FUNCTION_BLOCK "SINA_PARA_S"   // FB287, SCL
TITLE = 'one parameter exchange between SINAMICS and S7'
{ S7_Optimized_Access := 'TRUE' }
AUTHOR : DRVDPS7
FAMILY : DRIVES
NAME : SINA_PAS
VERSION : 5.0
// Copyright (C) Siemens AG 2012. All Rights Reserved. Confidential
// --------------------------------------------------------------------------- 
// SINA_PARA_S: Austausch eines beliebigen Parameter zwischen SINAMICS S120/G120 <-> S7
// -------------------------------------------------------------------------- Ersteller: J.B. Typical Team               Datum:  25.06.14        Vers.:3.0
//     Übernahme vom SINA_PARA Verion 2.9 und Abänderung zu SINA_PARA_S
//     Austausch nur noch eines Parameters
// 
// Änderung:  J.B. Typical Team                       08.07.14              3.1
//     Fehlerkorrektur und Initialisierung 
//     Änderung
// Änderung:  J.B. Typical Team                       30.07.14              4.0
//     Festlegung auf einheitlicher neuer Version 4.0
// 
// Änderung:  G.F. Typical Team                       20.05.15              4.1
//     Fehler bei der Umrechnung der Parameterwerte behoben
// 
// Änderung:  G.F. Typical Team                       15.09.15              4.2
//     Defaultwert des Parameters AxisNo von 0 auf 1 geändert
// 
// Änderung:  G.F. Typical Team                       06.10.15              4.3
//     Defaultwert des Parameters Done von 0 auf 1 geändert
// 
// Änderung:  J.B. Typical Team                       08.12.15              4.4
//     1. Wenn beim Parameter "Lesen" ein Fehler zurück gemeldet wird, 
//     soll das "Schreiben" abgebrochen werden
// 
//     2. Für den Datentyp DWORD mit/ohne Vorzeichen neuer Ablageort
//     (statt REAL nun DINT)
// 
//     3. Neue Ausgangsvariable Ready = Lesen/Schreiben der Parameter
//     abgeschlossen
// 
//     4. Austauch der Parameter kann jetzt abgebrochen werden
// 
//     5. Warnung durch Initialisierung elimininiert
// 
//     6. Eingang Laddr in hardwareId umbenannt
// 
// Änderung:  G.F. Typical Team                       24.11.16              4.5
//     - Fehlerausgabe bei unbekannten Datentyp (ErrorId := 5)
//     - Datentyp 10 (OctetString) wird unterstützt
//     - Datentyp 13 (TimeDifference) wird unterstützt
//     - Fehler bei Auftrag abbrechen behoben
// 
// Änderung:  G.F. Typical Team                       11.01.17              5.0
//     - Festlegung auf einheitlicher neuer Version 5.0 
// 
// Bibliothek V7
// Funktion: Austausch eines beliebigen Parameter zwischen SINAMICS S120/G120 <-> S7
// ********************************************************************************************************************************************************
// ************************************************************************FB283***************************************************************************
// ********************************************************************************************************************************************************
   VAR_INPUT
      Start : Bool := 0;   // Start command for read or write parameter / 0-->1 Start des gewählten azyklischen Auftrags
      ReadWrite : Bool := 0;   // Type of job 0 = read parameter, 1 = write parameter / 0 = Lesen; 1 = Schreiben
      Parameter : Int := 1;   // Number of parameter (number 1..65535) / Parameternummer
      Index : Int := 0;   // Subindex (number 0..65535) / Subindex (Number 1..65535)
      ValueWrite1 : Real := 0.0;   // Value of the write parameter (byte, word, float) / Schreibwert vom Typ REAL
      ValueWrite2 : DInt := 0;   // Value of the write parameter (dint) / Schreibwert vom Typ DINT32
      AxisNo : Byte := 16#01;   // Object ID of drive / Antriebsnummer
      hardwareId : HW_IO := 0;   // Configured diagnosis address of the module (DEC) for WRREC and RDREC Output variables / Hardware Identifer des Modul Acces Points / Istwertslots des zyklsichen Telegramms
   END_VAR
   VAR_OUTPUT
      Ready : Bool := 0;   // Read or write parameter order ready / Bereitschaftsrückmeldung für den Betrieb mit LAcycCom Bausteinen
      Busy : Bool := 0;   // Mode of operation is explained
      Done : Bool := 1;   // Mode of operation without mistake finishes
      ValueRead1 : Real := 0.0;   // Value of the read parameter (byte, word, float) / Gelesener Wert im Format REAL
      ValueRead2 : DInt := 0;   // Value of the read parameter (dint) / Gelesener Wert im Format DINT32
      Format : Byte := 16#00;   // Format of the value (Format 0x40..0x44) / Rückmeldung des Formats des gelesenen Parameters
      ErrorNo : Word := 16#0000;   // Error number (see table below) / Fehlernummer nach Profidrive Profil
      Error : Bool := 0;   // Error or faults are active / 1 = Anzeige eines aufgetretenen Fehlers
      ErrorId : DWord := 0;   // Mode of operation disturbance
      DiagId : Word := 16#0000;   // Extended communication error Static variables / Rückmeldeausgang der Systemfunktionen im Fehlerfall
   END_VAR
   VAR
      sbWrError : Bool := 0;   // Error when writing with SFB WRREC
      sbWrDone : Bool := 0;   // Data record written with SFB WRREC
      sbRdError : Bool := 0;   // Error when reading with SFB RDREC
      sbWrBusy : Bool := 0;   // Write Task busy SFB 53 WRREC sind beschäftigt
      sbRdBusy : Bool := 0;   // Read Task busy SFB 52 RDREC sind beschäftigt
      sbWrStart : Bool := 0;   // Start write job
      sbRdStart : Bool := 0;   // Start read job
      sbWrStart1 : Bool := 0;   // Start write job (first part of write commando)
      sbRdStart1 : Bool := 0;   // Start read job (first part of read commando)
      sbWrStart2 : Bool := 0;   // Start write job (second part of write commando)
      sbRdStart2 : Bool := 0;   // Start read job (second part of read commando)
      sbStart : Bool := 0;   // Positive edge of Start commando
      sbReady : Bool := 0;   // Positive edge of Ready
      sbRead : Bool := 0;   // Commando "Read"
      sbWrite : Bool := 0;   // Commando "Write"
      sbParaNo : Bool := 0;   // The count of parameter are Okay
      sbBusy : Bool := 0;   // Mode of operation is explained
      sbError : Bool := 0;   // Error or faults are active
      sbDone : Bool := 0;   // Job finished
      syFormat : Byte := 16#00;   // Format of the value (Format 0x40..0x44)
      syAxisNo : Byte := 0;   // Antriebsobjekt ID
      siReqRef : Int := 0;   // Reference number of request
      siErrorId : Int := 0;   // Function block fault Id
      siErrorCount : Int := 0;   // temporary error counter of retry job
      siMaxErrCount : Int := 12500;   // max. temporary error counter
      swParaError : Word := WORD#16#0000;   // Error of parameter
      sxReqParaMulti : Struct   // Telegramm for request/change parameter value, multi-parameter
         sxHeader : Struct   // Request header
            syReqRef : Byte := 16#00;   // Request reference (Request ID, mirrored in response)
            syReqId : Byte := 16#01;   // Request ID 0x1=Read
            syAxisNo : Byte := 16#00;   // Axis (0x0=Axis A | 0x1=Axis B)
            syParaNo : Byte := 16#00;   // No. of parameters (DEC: for single parameters=1)
         END_STRUCT;
         sxParaAdress : Struct   // Parameter address
            syAttr : Byte := 16#10;   // Attribute of parameters (0x10=Value, 0x30=Text)
            syElemNo : Byte := 16#01;   // No. of elements (DEC: for single elements=1)
            siParaNo : Int := 0;   // Number of parameter (Number 1..65535)
            siIndex : Int := 0;   // Subindex (Number 1..65535)
         END_STRUCT;
      END_STRUCT;
      sxChaParaMulti : Struct   // Telegramm for change parameter value, multi-parameter
         sxHeader : Struct   // Request header
            syReqRef : Byte := 16#00;   // Request reference (Request ID, mirrored in response)
            syReqId : Byte := 16#02;   // Request ID 0x2=Write
            syAxisNo : Byte := 16#00;   // Axis (0x0=Axis A | 0x1=Axis B)
            syParaNo : Byte := 16#00;   // No. of parameters (DEC: for single parameters=1)
         END_STRUCT;
         sxData : Array[1..12] of Byte;   // Parameter address (Attribute/Value (BYTE), Number of Elements (BYTE), Parameter number (2 BYTES), Subindex (2 BYTES),Parameter value (Format/Error (BYTE), Number of Values/Value of Error (BYTE), Value (BYTE or WORD or DWORD)
      END_STRUCT;
      sxRespParaMulti : Struct   // Telegramm for response parameter value, multi-parameter
         sxHeader : Struct   // Request header
            syReqRef : Byte := 16#00;   // Request reference (Request ID, mirrored in response)
            syReqId : Byte := 16#00;   // Request ID (0x1=Read | 0x2=Write)
            syAxisNo : Byte := 16#00;   // Axis (0x0=Axis A | 0x1=Axis B)
            syParaNo : Byte := 16#00;   // No. of parameters (DEC: for single parameters=1)
         END_STRUCT;
         sxData : Array[1..6] of Byte;   // Parameter value (Format/Error (BYTE), Number of Values/Value of Error (BYTE), Value (BYTE or WORD or DWORD)
      END_STRUCT;
      RDREC_1 : RDREC;
      WRREC_1 : WRREC;
      siLenHeader : Int := 4;   // Length of telegram of header
      siLenParaMulti : Int := 6;   // Length of telegram of data for request and response
      siLenChaPara : Int := 12;   // Length of telegram of data for change parameter Temporary variables
   END_VAR
   VAR_TEMP
      piCount : Int;   // Freely available counter variable
      piPointer : Int;   // Freely available pointer array variable
      piLenTele : Int;   // Length of telegram of buffer
      piRetSFC : Int;   // Status for fault analysis
      pwWordHigh : Word;   // Help variable of word
      pwWordLow : Word;   // Help variable of word
      pwWord1 : Word;   // Help variable of word
      pwWord2 : Word;   // Help variable of word
      pdDWordHigh : DWord;   // Help variable of dword
      pdDWordLow : DWord;   // Help variable of dword
      pdStatus : DWord;   // Status[1] = Error => Status[2] Error Decode + Status[3] Error Code
      pbValidSFB : Bool;   // Status SFB
      piLenSFB : UInt;   // Status length for SFB call
      pwErrorNo : Word;   // Error number
   END_VAR
BEGIN

   //=============================================================================
   //SIEMENS AG
   //(c)Copyright 2017 All Rights Reserved
   //-----------------------------------------------------------------------------
   // Library: DriveLib
   // Tested with: S7-1516-3 PN/DP V1.8
   // Engineering: TIA Portal V14
   // Restrictions: -
   // Requirements: S7-1200 / S7-1500
   // Functionality: read and write one parameter from/to a Sinamics
   //
   //=============================================================================

   // Auftrag "Parameter lesen" bzw. Auftrag "Parameter schreiben" wird nicht mehr ausgeführt
   IF NOT #sbBusy THEN
     #sbParaNo := TRUE;
     #syAxisNo := #AxisNo;
   END_IF;

   // Starten 
   IF #Start AND NOT #sbStart AND NOT #sbBusy THEN

     #sbReady := False;
     #sbError := False;
     #sbBusy := False;

     // Auftrag "Parameter lesen" erkennen
     IF NOT #ReadWrite THEN
       #sbRead := True;
       #sbWrStart := True;
       #sbRdStart := False;

       #sbWrite := False;
       #sbWrStart1 := False;
       #sbRdStart1 := False;
       #sbWrStart2 := False;
       #sbRdStart2 := False;

       // Referenzauftragsnummer erzeugen
       #siReqRef := #siReqRef + 1;

       // bei Überschreitung wieder zurücksetzen und von vorne (Wertebereich von 0-255)
       IF #siReqRef > 255 THEN
         #siReqRef := 0;
       END_IF;

       // Auftrag "Parameter schreiben" erkennen
     ELSE
       #sbWrite := True;
       #sbWrStart1 := True;
       #sbRdStart1 := False;
       #sbWrStart2 := False;
       #sbRdStart2 := False;

       #sbRead := False;
       #sbWrStart := False;
       #sbRdStart := False;

       // Referenzauftragsnummer erzeugen
       #siReqRef := #siReqRef + 1;

       // bei Überschreitung wieder zurücksetzen und von vorne (Wertebereich von 0-255)
       IF #siReqRef > 255 THEN
         #siReqRef := 0;
       END_IF;
     END_IF;

     // Fehler 4 und 5 wieder zurücknehmen
     IF (#siErrorId = 4) OR (#siErrorId = 5) THEN
       #sbError := False;
       #siErrorId := 0;
     END_IF;
   END_IF;

   // "Start commando" Flanke merken
   #sbStart := #Start;

   // Abbrechen
   IF NOT #Start THEN

     #siErrorCount := 0;
     // Schreib - oder Lesevorgang abbrechen
     #sbRead := False;
     #sbWrStart := False;
     #sbRdStart := False;

     #sbWrite := False;
     #sbWrStart1 := False;
     #sbRdStart1 := False;
     #sbWrStart2 := False;
     #sbRdStart2 := False;

     // Auftag ist noch beschäftigt => Fehler ausgeben
     IF #sbBusy THEN
       #sbError := True;
       #siErrorId := 4;
       #sbBusy := False;
     END_IF;
   END_IF;


   // Auftrag "Parameter lesen" wurde ausgelöst
   IF #sbParaNo AND #sbRead AND NOT #sbWrite THEN

     // Auftrag "Parameter lesen" vorbereiten und abschicken
     IF #sbWrStart THEN

       // Ablöschen des Sendepuffers
       // Parameternummer des Parameters 
       #sxReqParaMulti.sxParaAdress.siParaNo := 0;

       // Subindex des Parameters
       #sxReqParaMulti.sxParaAdress.siIndex := 0;

       // Auftrags-HEADER erstellen
       // Auftragsreferenz
       #sxReqParaMulti.sxHeader.syReqRef := INT_TO_BYTE(#siReqRef);

       // Auftragskennung 0x01=Request Parameters
       #sxReqParaMulti.sxHeader.syReqId := B#16#01;

       // Achse
       #sxReqParaMulti.sxHeader.syAxisNo := #syAxisNo;

       // Anzahl Parameter        
       #sxReqParaMulti.sxHeader.syParaNo := B#16#01;

       // Auftrags-PARAMETERADRESSE erstellen
       // Parameternummer des Parameters                                
       #sxReqParaMulti.sxParaAdress.siParaNo := #Parameter;

       // Subindex des Parameters
       #sxReqParaMulti.sxParaAdress.siIndex := #Index;

       // SCHREIBEN AZYKLISCH
       #piLenTele := #siLenHeader + #siLenParaMulti;
       #WRREC_1(REQ := True,                                // Startimpuls
                ID := #hardwareId,                         // Diagnoseadresse
                INDEX := 47,                                  // Rahmentyp
                LEN := INT_TO_UINT(#piLenTele),             // maximale Länge
                DONE => #sbWrDone,                           // Schreibauftrag beendet
                BUSY => #sbWrBusy,                           // Slave beschäftigt
                ERROR => #sbWrError,                          // Fehler beim Schreiben
                STATUS => #pdStatus,                           // Status[1] = Error => Status[2] Error Decode + Status[3] Error Code
                RECORD := #sxReqParaMulti);                    // Zeiger auf zu schreibenen Datensatzes

       // Ausgänge setzen
       #sbBusy := #sbWrBusy;
       #sbDone := #sbWrDone;

       // Fehler auswerten
       IF #sbWrError THEN

         // Fehlerstatus aus dem Doppelwort filtern und weitergeben                
         #pwWord1 := DWORD_TO_WORD(SHR(IN := (#pdStatus AND DW#16#FFFF00), N := 8));

         // Fehlerstatus setzen
         #siErrorId := 3;
         #DiagId := #pwWord1;

         //Temporärer Fehler: #pdStatus = 80A7, 80B5, 80C0, 80C1, 80C2, 80C3 oder 80C4 zulassen und nocheinmal versuchen
         IF NOT (#pwWord1 = DW#16#80A7) AND NOT (#pwWord1 = DW#16#80B5) AND NOT (#pwWord1 = DW#16#80C0) AND
           NOT (#pwWord1 = DW#16#80C1) AND NOT (#pwWord1 = DW#16#80C2) AND NOT (#pwWord1 = DW#16#80C3) AND
           NOT (#pwWord1 = DW#16#80C4) THEN

           // Wiederholungsauftrag wieder zurücknehmen 
           #sbWrStart := False;
           #sbRdStart := False;
           #sbRead := False;

           // Fehler ausgeben 
           #sbError := #sbWrError;

         ELSE
           // Fehlerwiederholauftrag ??                   
           IF #siErrorCount = #siMaxErrCount THEN

             // Wiederholungsauftrag wieder zurücknehmen
             #sbWrStart := False;
             #sbRdStart := False;
             #sbRead := False;

             //Fehlerzähler zurücksetzen
             #siErrorCount := 0;


             // Fehler ausgeben 
             #sbError := #sbWrError;

             // nix tun bis Zähler überläuft
           ELSE
             #siErrorCount := #siErrorCount + 1;
           END_IF;
         END_IF;

         // kein Fehler beim SCHEIBEN AZYKLISCH und Auftrag fertig 
       ELSIF NOT #sbWrBusy AND #sbWrDone THEN

         // Fehlerkennung zurücknehmen
         IF #siErrorId = 3 THEN
           #siErrorId := 0;
           #sbError := False;
         END_IF;

         #DiagId := W#16#00;

         // Schreibauftrag fertig melden und Leseantrag anstossen
         #sbWrStart := False;
         #sbRdStart := True;
       END_IF;
     END_IF; // Auftrag "Parameter lesen" vorbereiten und abschicken

     // vom Auftrag "Parameter lesen" die Antwort abwarten und dann auswerten
     IF #sbRdStart THEN

       // Ablöschen des Empfangspuffers
       #sxRespParaMulti.sxHeader.syReqRef := B#16#00;
       #sxRespParaMulti.sxHeader.syReqId := B#16#00;
       #sxRespParaMulti.sxHeader.syAxisNo := B#16#00;
       #sxRespParaMulti.sxHeader.syParaNo := B#16#00;

       FOR #piCount := 1 TO #siLenParaMulti DO
         #sxRespParaMulti.sxData[#piCount] := B#16#00;
       END_FOR;

       // LESEN AZYKLISCH
       #piLenTele := #siLenHeader + #siLenParaMulti;
       #RDREC_1(REQ := True,                                // Startimpuls
                ID := #hardwareId,                         // Diagnoseadresse        
                INDEX := 47,                                  // Rahmentyp           
                MLEN := INT_TO_UINT(#piLenTele),             // maximale Länge
                VALID => #pbValidSFB,                         // neuer Datensatz empfangen und gültig   
                BUSY => #sbRdBusy,                           // Slave beschäftigt
                ERROR => #sbRdError,                          // Fehler beim Schreiben
                STATUS => #pdStatus,                           // Status[1] = Error => Status[2] Error Decode + Status[3] Error Code 
                LEN => #piLenSFB,                           // Länge des gelesenen Datensatzes
                RECORD := #sxRespParaMulti);                   // Zeiger auf gelesenen Datensatz

       // Ausgänge setzen
       #sbBusy := #sbRdBusy;
       #sbDone := #pbValidSFB;

       // Fehler auswerten
       IF #sbRdError THEN
         // Fehlerstatus aus dem Doppelwort filtern und weitergeben                
         #pwWord1 := DWORD_TO_WORD(SHR(IN := (#pdStatus AND DW#16#FFFF00), N := 8));

         // Fehlerstatus setzen
         #siErrorId := 3;
         #DiagId := #pwWord1;

         //Temporärer Fehler: #pdStatus = 80A7, 80B5, 80C0, 80C1, 80C2, 80C3 oder 80C4 zulassen und nocheinmal versuchen
         IF NOT (#pwWord1 = DW#16#80A7) AND NOT (#pwWord1 = DW#16#80B5) AND NOT (#pwWord1 = DW#16#80C0) AND
           NOT (#pwWord1 = DW#16#80C1) AND NOT (#pwWord1 = DW#16#80C2) AND NOT (#pwWord1 = DW#16#80C3) AND
           NOT (#pwWord1 = DW#16#80C4) THEN

           // Wiederholungsauftrag wieder zurücknehmen  
           #sbWrStart := False;
           #sbRdStart := False;
           #sbRead := False;

           // Fehler ausgeben 
           #sbError := #sbRdError;

         ELSE
           // Fehlerwiederholauftrag ??                   
           IF #siErrorCount = #siMaxErrCount THEN

             // Wiederholungsauftrag wieder zurücknehmen
             #sbWrStart := False;
             #sbRdStart := False;
             #sbRead := False;

             //Fehlerzähler zurücksetzen
             #siErrorCount := 0;


             // Fehler ausgeben 
             #sbError := #sbRdError;

             // nix tun bis Zähler überläuft
           ELSE
             #siErrorCount := #siErrorCount + 1;
           END_IF;
         END_IF;

         // Fehler : die Auftragsreferenz der Antwort übertimmt nicht mit der Auftragsreferenz der Anfrage überein
       ELSIF NOT (#siReqRef = BYTE_TO_INT(#sxRespParaMulti.sxHeader.syReqRef)) AND NOT #sbRdBusy AND #pbValidSFB THEN
         #siErrorId := 1;
         #sbError := True;
         #sbDone := False;

         // Wiederholungsauftrag wieder zurücknehmen  
         #sbWrStart := False;
         #sbRdStart := False;
         #sbRead := False;

         // Fehler : falsche Auftragskennung zurück erhalten    
       ELSIF NOT (#sxRespParaMulti.sxHeader.syReqId = B#16#81 OR #sxRespParaMulti.sxHeader.syReqId = B#16#01) AND
         NOT #sbRdBusy AND #pbValidSFB THEN
         #siErrorId := 1;
         #sbError := True;
         #sbDone := False;

         // Wiederholungsauftrag wieder zurücknehmen  
         #sbWrStart := False;
         #sbRdStart := False;
         #sbRead := False;

         // Fehler : die angeforderte Anzahl Parameter entspricht nicht der übermittelten Anzahl Parameter überein
       ELSIF NOT (#sxRespParaMulti.sxHeader.syParaNo = B#16#01) AND NOT #sbRdBusy AND #pbValidSFB THEN
         #siErrorId := 1;
         #sbError := True;
         #sbDone := False;

         // Wiederholungsauftrag wieder zurücknehmen  
         #sbWrStart := False;
         #sbRdStart := False;
         #sbRead := False;

         // Fehler : die Achse entspricht nicht der übergebenen Achse
       ELSIF NOT (#syAxisNo = #sxRespParaMulti.sxHeader.syAxisNo) AND NOT #sbRdBusy AND #pbValidSFB THEN
         #siErrorId := 1;
         #sbError := True;
         #sbDone := False;

         // Wiederholungsauftrag wieder zurücknehmen  
         #sbWrStart := False;
         #sbRdStart := False;
         #sbRead := False;

         // kein Fehler beim LESEN AZYKLISCH und Auftrag fertig 
       ELSIF NOT #sbRdBusy AND #pbValidSFB THEN

         // die angefragten Parameter auswerten und im Puffer abspeichern

         // ermitteltes Format des Parameters abspeichern
         #syFormat := #sxRespParaMulti.sxData[1];

         // Format = Error ? = > gesendeter Parameter fehlerhaft
         IF (BYTE_TO_INT(#sxRespParaMulti.sxData[1]) = 68) THEN

           // Format = Error, zwei Bytes zu übermittelten Fehlernummer zusammenfassen
           #pwWordHigh := SHL(IN := BYTE_TO_WORD(#sxRespParaMulti.sxData[3]), N := 8);
           #pwWordLow := BYTE_TO_WORD(#sxRespParaMulti.sxData[4]);

           #sbError := True;

           // ermittelte Fehlernummer im Puffer abspeichern
           #ErrorNo := #pwWordHigh XOR #pwWordLow;

           // Die Fehlerhaftigkeit des erkannten Parameter in der Fehlernummer eintragen   
           #swParaError := #swParaError OR W#16#01;

           // Format = Byte ? = > gesendeter Parameter ein Byte lang ohne Vorzeichen
         ELSIF (#sxRespParaMulti.sxData[1] = B#16#41) OR (#sxRespParaMulti.sxData[1] = B#16#05) THEN

           // ermittelter Parameterwert eintragen (Byte) 
           #ValueRead1 := USINT_TO_REAL(BYTE_TO_USINT(#sxRespParaMulti.sxData[3]));
           #ValueRead2 := 0;

           // ermittelte Fehlernummer im Puffer zurücksetzen
           #ErrorNo := W#16#00;

           // Die Fehlerhaftigkeit des erkannten Parameter in der Fehlernummer löschen   
           #swParaError := #swParaError AND W#16#FFFE;

           // Format = Byte ? = > gesendeter Parameter ein Byte lang mit Vorzeichen
         ELSIF (#sxRespParaMulti.sxData[1] = B#16#02) THEN

           // ermittelter Parameterwert eintragen (Byte) 
           #ValueRead1 := SINT_TO_REAL(BYTE_TO_SINT(#sxRespParaMulti.sxData[3]));
           #ValueRead2 := 0;

           // ermittelte Fehlernummer im Puffer zurücksetzen
           #ErrorNo := W#16#00;

           // Die Fehlerhaftigkeit des erkannten Parameter in der Fehlernummer löschen   
           #swParaError := #swParaError AND W#16#FFFE;

           // Format = Word ? = > gesendeter Parameter zwei Bytes lang ohne Vorzeichen
         ELSIF (#sxRespParaMulti.sxData[1] = B#16#42) OR (#sxRespParaMulti.sxData[1] = B#16#06)
           OR (#sxRespParaMulti.sxData[1] = B#16#0A) THEN

           // Format = Word, zwei Bytes zu übermitteltem Parameterwert zusammenfassen
           #pwWordHigh := SHL(IN := BYTE_TO_WORD(#sxRespParaMulti.sxData[3]), N := 8);
           #pwWordLow := BYTE_TO_WORD(#sxRespParaMulti.sxData[4]);
           #pwWord1 := #pwWordHigh XOR #pwWordLow;

           // ermittelter Parameterwert eintragen (Word)
           #ValueRead1 := UINT_TO_REAL(WORD_TO_UINT(#pwWord1));
           #ValueRead2 := 0;

           // ermittelte Fehlernummer im Puffer zurücksetzen
           #ErrorNo := W#16#00;

           // Die Fehlerhaftigkeit des erkannten Parameter in der Fehlernummer löschen   
           #swParaError := #swParaError AND W#16#FFFE;

           // Format = Word ? = > gesendeter Parameter zwei Bytes lang mit Vorzeichen
         ELSIF (#sxRespParaMulti.sxData[1] = B#16#03) THEN

           // Format = Word, zwei Bytes zu übermitteltem Parameterwert zusammenfassen
           #pwWordHigh := SHL(IN := BYTE_TO_WORD(#sxRespParaMulti.sxData[3]), N := 8);
           #pwWordLow := BYTE_TO_WORD(#sxRespParaMulti.sxData[4]);
           #pwWord1 := #pwWordHigh XOR #pwWordLow;

           // ermittelter Parameterwert eintragen (Word)
           #ValueRead1 := INT_TO_REAL(WORD_TO_INT(#pwWord1));
           #ValueRead2 := 0;

           // ermittelte Fehlernummer im Puffer zurücksetzen
           #ErrorNo := W#16#00;

           // Die Fehlerhaftigkeit des erkannten Parameter in der Fehlernummer löschen   
           #swParaError := #swParaError AND W#16#FFFE;

           // Format = Double Word ? = > gesendeter Parameter vier Bytes lang ohne Vorzeichen
         ELSIF (#sxRespParaMulti.sxData[1] = B#16#43) OR (#sxRespParaMulti.sxData[1] = B#16#07) OR
           (#sxRespParaMulti.sxData[1] = B#16#0D) THEN

           // Format = Double Word, vier Bytes zu übermitteltem Parameterwert zusammenfassen
           #pwWordHigh := SHL(IN := BYTE_TO_WORD(#sxRespParaMulti.sxData[3]), N := 8);
           #pwWordLow := BYTE_TO_WORD(#sxRespParaMulti.sxData[4]);
           #pwWord1 := #pwWordHigh XOR #pwWordLow;

           #pwWordHigh := SHL(IN := BYTE_TO_WORD(#sxRespParaMulti.sxData[5]), N := 8);
           #pwWordLow := BYTE_TO_WORD(#sxRespParaMulti.sxData[6]);
           #pwWord2 := #pwWordHigh XOR #pwWordLow;

           #pdDWordHigh := SHL(IN := WORD_TO_DWORD(#pwWord1), N := 16);
           #pdDWordLow := WORD_TO_DWORD(#pwWord2);

           // ermittelter Parameterwert eintragen (Word)
           #ValueRead1 := 0.0;
           #ValueRead2 := DWORD_TO_DINT(#pdDWordHigh XOR #pdDWordLow);

           // ermittelte Fehlernummer im Puffer zurücksetzen
           #ErrorNo := W#16#00;

           // Die Fehlerhaftigkeit des erkannten Parameter in der Fehlernummer löschen   
           #swParaError := #swParaError AND W#16#FFFE;

           // Format = Double Word ? = > gesendeter Parameter vier Bytes lang mit Vorzeichen
         ELSIF (#sxRespParaMulti.sxData[1] = B#16#04) THEN

           // Format = Double Word, vier Bytes zu übermitteltem Parameterwert zusammenfassen
           #pwWordHigh := SHL(IN := BYTE_TO_WORD(#sxRespParaMulti.sxData[3]), N := 8);
           #pwWordLow := BYTE_TO_WORD(#sxRespParaMulti.sxData[4]);
           #pwWord1 := #pwWordHigh XOR #pwWordLow;

           #pwWordHigh := SHL(IN := BYTE_TO_WORD(#sxRespParaMulti.sxData[5]), N := 8);
           #pwWordLow := BYTE_TO_WORD(#sxRespParaMulti.sxData[6]);
           #pwWord2 := #pwWordHigh XOR #pwWordLow;

           #pdDWordHigh := SHL(IN := WORD_TO_DWORD(#pwWord1), N := 16);
           #pdDWordLow := WORD_TO_DWORD(#pwWord2);

           // ermittelter Parameterwert eintragen (Word)
           #ValueRead1 := 0.0;
           #ValueRead2 := DWORD_TO_DINT(#pdDWordHigh XOR #pdDWordLow);

           // ermittelte Fehlernummer im Puffer zurücksetzen
           #ErrorNo := W#16#00;

           // Die Fehlerhaftigkeit des erkannten Parameter in der Fehlernummer löschen   
           #swParaError := #swParaError AND W#16#FFFE;

           // Format = Double Word ? = > gesendeter Parameter vier Bytes lang (FloatingPoint)
         ELSIF (#sxRespParaMulti.sxData[1] = B#16#08) THEN

           // Format = Double Word, vier Bytes zu übermitteltem Parameterwert zusammenfassen
           #pwWordHigh := SHL(IN := BYTE_TO_WORD(#sxRespParaMulti.sxData[3]), N := 8);
           #pwWordLow := BYTE_TO_WORD(#sxRespParaMulti.sxData[4]);
           #pwWord1 := #pwWordHigh XOR #pwWordLow;

           #pwWordHigh := SHL(IN := BYTE_TO_WORD(#sxRespParaMulti.sxData[5]), N := 8);
           #pwWordLow := BYTE_TO_WORD(#sxRespParaMulti.sxData[6]);
           #pwWord2 := #pwWordHigh XOR #pwWordLow;

           #pdDWordHigh := SHL(IN := WORD_TO_DWORD(#pwWord1), N := 16);
           #pdDWordLow := WORD_TO_DWORD(#pwWord2);

           // ermittelter Parameterwert eintragen (Word)
           #ValueRead1 := DWORD_TO_REAL(#pdDWordHigh XOR #pdDWordLow);
           #ValueRead2 := 0;

           // ermittelte Fehlernummer im Puffer zurücksetzen
           #ErrorNo := W#16#00;

           // Die Fehlerhaftigkeit des erkannten Parameter in der Fehlernummer löschen   
           #swParaError := #swParaError AND W#16#FFFE;

           // Unbekanter Datentyp
         ELSE

           #siErrorId := 5;
           #sbError := True;
           #sbDone := False;
           // Die Fehlerhaftigkeit des erkannten Parameter in der Fehlernummer eintragen   
           #swParaError := #swParaError OR W#16#01;

         END_IF;

         // Fehlerkennung zurücknehmen
         IF (#siErrorId = 3) OR (#siErrorId = 1) THEN
           #siErrorId := 0;
           #sbError := False;
         END_IF;

         #DiagId := W#16#00;

         // Auftrag : Parameter lesen ist abgeschlossen
         #sbRdStart := False;
         #sbRead := False;
       END_IF; // kein Fehler beim LESEN AZYKLISCH und Auftrag fertig 
     END_IF; // vom Auftrag "Parameter lesen" die Antwort abwarten und dann auswerten 
   END_IF; // Auftrag "Parameter lesen" wurde ausgelöst

   // Auftrag "Parameter schreiben" wurde ausgelöst
   IF #sbParaNo AND NOT #sbRead AND #sbWrite THEN

     // Auftrag "Parameter schreiben" bzw. "ändern" besteht aus zwei Aufträgen
     // 1. Teilauftrag "Parameter lesen"
     // 2. Teilauftrag "Parameter schreiben bzw. ändern"

     // 1. Teilauftrag "Parameter lesen" vorbereiten und abschicken
     IF #sbWrStart1 THEN

       // Ablöschen des Sendepuffers
       // Parameternummer des Parameters 
       #sxReqParaMulti.sxParaAdress.siParaNo := 0;

       // Subindex des Parameters
       #sxReqParaMulti.sxParaAdress.siIndex := 0;

       // Auftrags-HEADER erstellen
       // Auftragsreferenz
       #sxReqParaMulti.sxHeader.syReqRef := INT_TO_BYTE(#siReqRef);

       // Auftragskennung 0x01=Request Parameters
       #sxReqParaMulti.sxHeader.syReqId := B#16#01;

       // Achse
       #sxReqParaMulti.sxHeader.syAxisNo := #syAxisNo;

       // Anzahl Parameter        
       #sxReqParaMulti.sxHeader.syParaNo := B#16#01;

       // Auftrags-PARAMETERADRESSE erstellen
       // Parameternummer des Parameters                                
       #sxReqParaMulti.sxParaAdress.siParaNo := #Parameter;

       // Subindex des Parameters
       #sxReqParaMulti.sxParaAdress.siIndex := #Index;

       // SCHREIBEN AZYKLISCH
       #piLenTele := #siLenHeader + #siLenParaMulti;
       #WRREC_1(REQ := True,                                // Startimpuls
                ID := #hardwareId,                         // Diagnoseadresse
                INDEX := 47,                                  // Rahmentyp
                LEN := INT_TO_UINT(#piLenTele),             // maximale Länge
                DONE => #sbWrDone,                           // Schreibauftrag beendet
                BUSY => #sbWrBusy,                           // Slave beschäftigt
                ERROR => #sbWrError,                          // Fehler beim Schreiben
                STATUS => #pdStatus,                           // Status[1] = Error => Status[2] Error Decode + Status[3] Error Code
                RECORD := #sxReqParaMulti);                    // Zeiger auf zu schreibenen Datensatz

       // Ausgänge setzen
       #sbBusy := #sbWrBusy;
       #sbDone := #sbWrDone;

       // Fehler auswerten
       IF #sbWrError THEN

         // Fehlerstatus aus dem Doppelwort filtern und weitergeben                
         #pwWord1 := DWORD_TO_WORD(SHR(IN := (#pdStatus AND DW#16#FFFF00), N := 8));

         // Fehlerstatus setzen
         #siErrorId := 3;
         #DiagId := #pwWord1;

         //Temporärer Fehler: #pdStatus = 80A7, 80B5, 80C0, 80C1, 80C2, 80C3 oder 80C4 zulassen und nocheinmal versuchen
         IF NOT (#pwWord1 = DW#16#80A7) AND NOT (#pwWord1 = DW#16#80B5) AND NOT (#pwWord1 = DW#16#80C0) AND
           NOT (#pwWord1 = DW#16#80C1) AND NOT (#pwWord1 = DW#16#80C2) AND NOT (#pwWord1 = DW#16#80C3) AND
           NOT (#pwWord1 = DW#16#80C4) THEN

           // Wiederholungsauftrag wieder zurücknehmen
           #sbWrStart1 := False;
           #sbRdStart1 := False;
           #sbWrite := False;

           // Fehler ausgeben 
           #sbError := #sbWrError;

         ELSE
           // Fehlerwiederholauftrag ??                   
           IF #siErrorCount = #siMaxErrCount THEN

             // Wiederholungsauftrag wieder zurücknehmen
             #sbWrStart1 := False;
             #sbRdStart1 := False;
             #sbWrite := False;

             //Fehlerzähler zurücksetzen
             #siErrorCount := 0;


             // Fehler ausgeben 
             #sbError := #sbWrError;
             // nix tun bis Zähler überläuft
           ELSE
             #siErrorCount := #siErrorCount + 1;
           END_IF;
         END_IF;

         // kein Fehler beim SCHEIBEN AZYKLISCH und Auftrag fertig 
       ELSIF NOT #sbWrBusy AND #sbWrDone THEN

         // Fehlerkennung zurücknehmen
         IF (#siErrorId = 3) THEN
           #siErrorId := 0;
           #sbError := False;
         END_IF;

         #DiagId := W#16#00;

         // Schreibauftrag fertig melden und Leseantrag anstossen
         #sbWrStart1 := False;
         #sbRdStart1 := True;
       END_IF;
     END_IF; // 1. Teilauftrag "Parameter lesen" vorbereiten und abschicken

     // vom 1. Teilauftrag "Parameter lesen" die Antwort abwarten und dann auswerten
     IF #sbRdStart1 THEN

       // Ablöschen des Empfangspuffers
       #sxRespParaMulti.sxHeader.syReqRef := B#16#00;
       #sxRespParaMulti.sxHeader.syReqId := B#16#00;
       #sxRespParaMulti.sxHeader.syAxisNo := B#16#00;
       #sxRespParaMulti.sxHeader.syParaNo := B#16#00;

       FOR #piCount := 1 TO #siLenParaMulti DO
         #sxRespParaMulti.sxData[#piCount] := B#16#00;
       END_FOR;

       // LESEN AZYKLISCH
       #piLenTele := #siLenHeader + #siLenParaMulti;
       #RDREC_1(REQ := True,                                // Startimpuls
                ID := #hardwareId,                         // Diagnoseadresse        
                INDEX := 47,                                  // Rahmentyp           
                MLEN := INT_TO_UINT(#piLenTele),             // maximale Länge
                VALID => #pbValidSFB,                         // neuer Datensatz empfangen und gültig      
                BUSY => #sbRdBusy,                           // Slave beschäftigt
                ERROR => #sbRdError,                          // Fehler beim Schreiben
                STATUS => #pdStatus,                           // Status[1] = Error => Status[2] Error Decode + Status[3] Error Code 
                LEN => #piLenSFB,                           // Länge des gelesenen Datensatzes
                RECORD := #sxRespParaMulti);                   // Zeiger auf gelesenen Datensatz

       // Ausgänge setzen
       #sbBusy := #sbRdBusy;
       #sbDone := #pbValidSFB;

       // Fehler auswerten
       IF #sbRdError THEN
         // Fehlerstatus aus dem Doppelwort filtern und weitergeben                
         #pwWord1 := DWORD_TO_WORD(SHR(IN := (#pdStatus AND DW#16#FFFF00), N := 8));

         // Fehlerstatus setzen
         #siErrorId := 3;
         #DiagId := #pwWord1;

         //Temporärer Fehler: #pdStatus = 80A7, 80B5, 80C0, 80C1, 80C2, 80C3 oder 80C4 zulassen und nocheinmal versuchen
         IF NOT (#pwWord1 = DW#16#80A7) AND NOT (#pwWord1 = DW#16#80B5) AND NOT (#pwWord1 = DW#16#80C0) AND
           NOT (#pwWord1 = DW#16#80C1) AND NOT (#pwWord1 = DW#16#80C2) AND NOT (#pwWord1 = DW#16#80C3) AND
           NOT (#pwWord1 = DW#16#80C4) THEN

           // Wiederholungsauftrag wieder zurücknehmen
           #sbWrStart1 := False;
           #sbRdStart1 := False;
           #sbWrite := False;

           // Fehler ausgeben 
           #sbError := #sbRdError;

         ELSE
           // Fehlerwiederholauftrag ??                   
           IF #siErrorCount = #siMaxErrCount THEN

             // Wiederholungsauftrag wieder zurücknehmen
             #sbWrStart1 := False;
             #sbRdStart1 := False;
             #sbWrite := False;

             //Fehlerzähler zurücksetzen
             #siErrorCount := 0;


             // Fehler ausgeben 
             #sbError := #sbRdError;

             // nix tun bis Zähler überläuft
           ELSE
             #siErrorCount := #siErrorCount + 1;
           END_IF;
         END_IF;

         // Fehler : die Auftragsreferenz der Antwort übertimmt nicht mit der Auftragsreferenz der Anfrage überein
       ELSIF NOT (#siReqRef = BYTE_TO_INT(#sxRespParaMulti.sxHeader.syReqRef)) AND NOT #sbRdBusy AND #pbValidSFB THEN
         #siErrorId := 1;
         #sbError := True;
         #sbDone := False;

         // Wiederholungsauftrag wieder zurücknehmen
         #sbWrStart1 := False;
         #sbRdStart1 := False;
         #sbWrite := False;

         // Fehler : falsche Auftragskennung zurück erhalten    
       ELSIF NOT (#sxRespParaMulti.sxHeader.syReqId = B#16#81 OR #sxRespParaMulti.sxHeader.syReqId = B#16#01) AND
         NOT #sbRdBusy AND #pbValidSFB THEN
         #siErrorId := 1;
         #sbError := True;
         #sbDone := False;

         // Wiederholungsauftrag wieder zurücknehmen
         #sbWrStart1 := False;
         #sbRdStart1 := False;
         #sbWrite := False;

         // Fehler : die angeforderte Anzahl Parameter entspricht nicht der übermittelten Anzahl Parameter überein
       ELSIF NOT (#sxRespParaMulti.sxHeader.syParaNo = B#16#01) AND NOT #sbRdBusy AND #pbValidSFB THEN
         #siErrorId := 1;
         #sbError := True;
         #sbDone := False;

         // Wiederholungsauftrag wieder zurücknehmen
         #sbWrStart1 := False;
         #sbRdStart1 := False;
         #sbWrite := False;

         // Fehler : die Achse entspricht nicht der übergebenen Achse
       ELSIF NOT (#syAxisNo = #sxRespParaMulti.sxHeader.syAxisNo) AND NOT #sbRdBusy AND #pbValidSFB THEN
         #siErrorId := 1;
         #sbError := True;
         #sbDone := False;

         // Wiederholungsauftrag wieder zurücknehmen
         #sbWrStart1 := False;
         #sbRdStart1 := False;
         #sbWrite := False;

         // kein Fehler beim LESEN AZYKLISCH und Auftrag fertig 
       ELSIF NOT #sbRdBusy AND #pbValidSFB THEN

         // die angefragten Parameter auswerten und im Puffer abspeichern
         // ermitteltes Format des Parameters abspeichern
         #syFormat := #sxRespParaMulti.sxData[1];

         // Format = Error ? = > gesendeter Parameter fehlerhaft
         IF (BYTE_TO_INT(#sxRespParaMulti.sxData[1]) = 68) THEN

           // Format = Error, zwei Bytes zu übermittelten Fehlernummer zusammenfassen
           #pwWordHigh := SHL(IN := BYTE_TO_WORD(#sxRespParaMulti.sxData[3]), N := 8);
           #pwWordLow := BYTE_TO_WORD(#sxRespParaMulti.sxData[4]);

           #sbError := True;

           // ermittelte Fehlernummer im Puffer abspeichern
           #ErrorNo := #pwWordHigh XOR #pwWordLow;

           // Die Fehlerhaftigkeit des erkannten Parameter in der Fehlernummer eintragen   
           #swParaError := #swParaError OR W#16#01;

           // Format = Byte ? = > gesendeter Parameter ein Byte lang
         ELSIF (#sxRespParaMulti.sxData[1] = B#16#41) OR
           (#sxRespParaMulti.sxData[1] = B#16#02) OR (#sxRespParaMulti.sxData[1] = B#16#05) THEN

           // ermittelte Fehlernummer im Puffer zurücksetzen
           #ErrorNo := W#16#00;

           // Die Fehlerhaftigkeit des erkannten Parameter in der Fehlernummer löschen   
           #swParaError := #swParaError AND W#16#FFFE;

           // Format = Word ? = > gesendeter Parameter zwei Bytes lang
         ELSIF (#sxRespParaMulti.sxData[1] = B#16#42) OR (#sxRespParaMulti.sxData[1] = B#16#03)
           OR (#sxRespParaMulti.sxData[1] = B#16#06) OR (#sxRespParaMulti.sxData[1] = B#16#0A) THEN

           // ermittelte Fehlernummer im Puffer zurücksetzen
           #ErrorNo := W#16#00;

           // Die Fehlerhaftigkeit des erkannten Parameter in der Fehlernummer löschen   
           #swParaError := #swParaError AND W#16#FFFE;


           // Format = Double Word ? = > gesendeter Parameter vier Bytes lang
         ELSIF (#sxRespParaMulti.sxData[1] = B#16#43) OR (#sxRespParaMulti.sxData[1] = B#16#04) OR
           (#sxRespParaMulti.sxData[1] = B#16#07) OR (#sxRespParaMulti.sxData[1] = B#16#08) OR
           (#sxRespParaMulti.sxData[1] = B#16#0D) THEN

           // ermittelte Fehlernummer im Puffer zurücksetzen
           #ErrorNo := W#16#00;

           // Die Fehlerhaftigkeit des erkannten Parameter in der Fehlernummer löschen   
           #swParaError := #swParaError AND W#16#FFFE;

           // Unbekanter Datentyp
         ELSE

           #siErrorId := 5;
           #sbError := True;
           #sbDone := False;
           // Die Fehlerhaftigkeit des erkannten Parameter in der Fehlernummer eintragen   
           #swParaError := #swParaError OR W#16#01;

         END_IF;

         // Fehlerkennung zurücknehmen
         IF (#siErrorId = 3) OR (#siErrorId = 1) THEN
           #siErrorId := 0;
           #sbError := False;
         END_IF;

         #DiagId := W#16#00;

         // 1. Teilauftrag "Parameter lesen" ist abgeschlossen
         #sbRdStart1 := False;

         // einer der gesendeten Parameter ist fehlerhaft => Abbruch, kein "Parameter schreiben" erforderlich
         IF (#swParaError = W#16#00) THEN
           #sbWrStart2 := True;
         ELSE
           #sbWrStart2 := False;
         END_IF;
       END_IF; // kein Fehler beim LESEN AZYKLISCH und Auftrag fertig 
     END_IF; // vom 1. Teilauftrag "Parameter lesen" die Antwort abwarten und dann auswerten 

     // 2. Teilauftrag "Parameter schreiben bzw. ändern" vorbereiten und abschicken
     IF #sbWrStart2 THEN

       // Ablöschen des Sendepuffers            
       FOR #piCount := 1 TO #siLenChaPara DO
         // Parameteradresse und Parameterwert des Parameters 
         #sxChaParaMulti.sxData[#piCount] := B#16#00;
       END_FOR;

       // Auftrags-HEADER erstellen
       // Auftragsreferenz
       #sxChaParaMulti.sxHeader.syReqRef := INT_TO_BYTE(#siReqRef);

       // Auftragskennung 0x01=Request Parameters | 0x02=Change Parameters
       #sxChaParaMulti.sxHeader.syReqId := B#16#02;

       // Achse
       #sxChaParaMulti.sxHeader.syAxisNo := #syAxisNo;

       // Anzahl Parameter        
       #sxChaParaMulti.sxHeader.syParaNo := B#16#01;

       // Auftrags-PARAMETERADRESSE erstellen                
       // Attribute of parameters (0x10=Value, 0x30=Text)
       #sxChaParaMulti.sxData[1] := B#16#10;

       // No. of elements (DEC: for single elements=1) 
       #sxChaParaMulti.sxData[2] := B#16#01;

       // Parameternummer des Parameters                                
       #sxChaParaMulti.sxData[4] := INT_TO_BYTE(#Parameter);
       #sxChaParaMulti.sxData[3] := WORD_TO_BYTE(SHR(IN := INT_TO_WORD(#Parameter), N := 8));

       // Subindex des Parameters
       #sxChaParaMulti.sxData[6] := INT_TO_BYTE(#Index);
       #sxChaParaMulti.sxData[5] := WORD_TO_BYTE(SHR(IN := INT_TO_WORD(#Index), N := 8));

       // Auftrags-PARAMETERVALUE erstellen    
       // Format (BYTE, WORD, DWORD des Parameterwert übergeben
       #sxChaParaMulti.sxData[7] := #syFormat;

       // Number of value
       #sxChaParaMulti.sxData[8] := B#16#01;

       // Value of parameter in Bytes
       IF (#syFormat = B#16#41) OR
         (#syFormat = B#16#02) OR (#syFormat = B#16#05) THEN

         #sxChaParaMulti.sxData[9] := WORD_TO_BYTE(DWORD_TO_WORD(DINT_TO_DWORD(REAL_TO_DINT(#ValueWrite1))));
         #sxChaParaMulti.sxData[10] := 16#00;  //WORD_TO_BYTE(DWORD_TO_WORD(SHR(IN := DINT_TO_DWORD(REAL_TO_DINT(#ValueWrite1)), N := 8)));

         // Value of parameter in Word
       ELSIF (#syFormat = B#16#42) OR (#syFormat = B#16#03) OR
         (#syFormat = B#16#06) OR (#syFormat = B#16#0A) THEN

         #sxChaParaMulti.sxData[10] := WORD_TO_BYTE(DWORD_TO_WORD(DINT_TO_DWORD(REAL_TO_DINT(#ValueWrite1))));
         #sxChaParaMulti.sxData[9] := WORD_TO_BYTE(DWORD_TO_WORD(SHR(IN := DINT_TO_DWORD(REAL_TO_DINT(#ValueWrite1)), N := 8)));

         // Value of parameter in DWord    
       ELSIF (#syFormat = B#16#43) OR (#syFormat = B#16#04) OR
         (#syFormat = B#16#07) OR (#syFormat = B#16#0D) THEN

         #sxChaParaMulti.sxData[12] := WORD_TO_BYTE(DWORD_TO_WORD(DINT_TO_DWORD(#ValueWrite2)));
         #sxChaParaMulti.sxData[11] := WORD_TO_BYTE(DWORD_TO_WORD(SHR(IN := DINT_TO_DWORD(#ValueWrite2), N := 8)));
         #sxChaParaMulti.sxData[10] := WORD_TO_BYTE(DWORD_TO_WORD(SHR(IN := DINT_TO_DWORD(#ValueWrite2), N := 16)));
         #sxChaParaMulti.sxData[9] := WORD_TO_BYTE(DWORD_TO_WORD(SHR(IN := DINT_TO_DWORD(#ValueWrite2), N := 24)));


         // Value of parameter in DWord (FloatingPoint)   
       ELSIF (#syFormat = B#16#08) THEN

         #sxChaParaMulti.sxData[12] := WORD_TO_BYTE(DWORD_TO_WORD(REAL_TO_DWORD(#ValueWrite1)));
         #sxChaParaMulti.sxData[11] := WORD_TO_BYTE(DWORD_TO_WORD(SHR(IN := REAL_TO_DWORD(#ValueWrite1), N := 8)));
         #sxChaParaMulti.sxData[10] := WORD_TO_BYTE(DWORD_TO_WORD(SHR(IN := REAL_TO_DWORD(#ValueWrite1), N := 16)));
         #sxChaParaMulti.sxData[9] := WORD_TO_BYTE(DWORD_TO_WORD(SHR(IN := REAL_TO_DWORD(#ValueWrite1), N := 24)));

       END_IF;

       // SCHREIBEN AZYKLISCH
       #piLenTele := #siLenHeader + #siLenChaPara;
       #WRREC_1(REQ := True,                                // Startimpuls
                ID := #hardwareId,                         // Diagnoseadresse
                INDEX := 47,                                  // Rahmentyp
                LEN := INT_TO_UINT(#piLenTele),             // maximale Länge
                DONE => #sbWrDone,                           // Schreibauftrag beendet
                BUSY => #sbWrBusy,                           // Slave beschäftigt
                ERROR => #sbWrError,                          // Fehler beim Schreiben
                STATUS => #pdStatus,                           // Status[1] = Error => Status[2] Error Decode + Status[3] Error Code
                RECORD := #sxChaParaMulti);                    // Zeiger auf zu schreibenen Datensatzes

       // Ausgänge setzen
       #sbBusy := #sbWrBusy;
       #sbDone := #sbWrDone;

       // Fehler auswerten
       IF #sbWrError THEN
         // Fehlerstatus aus dem Doppelwort filtern und weitergeben                
         #pwWord1 := DWORD_TO_WORD(SHR(IN := (#pdStatus AND DW#16#FFFF00), N := 8));

         // Fehlerstatus setzen
         #siErrorId := 3;
         #sbError := False;
         #DiagId := #pwWord1;

         //Temporärer Fehler: #pdStatus = 80A7, 80B5, 80C0, 80C1, 80C2, 80C3 oder 80C4 zulassen und nocheinmal versuchen
         IF NOT (#pwWord1 = DW#16#80A7) AND NOT (#pwWord1 = DW#16#80B5) AND NOT (#pwWord1 = DW#16#80C0) AND
           NOT (#pwWord1 = DW#16#80C1) AND NOT (#pwWord1 = DW#16#80C2) AND NOT (#pwWord1 = DW#16#80C3) AND
           NOT (#pwWord1 = DW#16#80C4) THEN

           // Wiederholungsauftrag wieder zurücknehmen
           #sbWrStart2 := False;
           #sbRdStart2 := False;
           #sbWrite := False;

           // Fehler ausgeben 
           #sbError := #sbWrError;

         ELSE
           // Fehlerwiederholauftrag ??                   
           IF #siErrorCount = #siMaxErrCount THEN

             // Wiederholungsauftrag wieder zurücknehmen
             #sbWrStart2 := False;
             #sbRdStart2 := False;
             #sbWrite := False;

             //Fehlerzähler zurücksetzen
             #siErrorCount := 0;


             // Fehler ausgeben 
             #sbError := #sbWrError;

             // nix tun bis Zähler überläuft
           ELSE
             #siErrorCount := #siErrorCount + 1;
           END_IF;
         END_IF;

         // kein Fehler beim SCHEIBEN AZYKLISCH und Auftrag fertig 
       ELSIF NOT #sbWrBusy AND #sbWrDone THEN
         // Fehlerkennung zurücknehmen
         #DiagId := W#16#00;

         // Schreibauftrag fertig melden und Leseantrag anstossen
         #sbWrStart2 := False;
         #sbRdStart2 := True;
       END_IF;
     END_IF; // 2. Teilauftrag "Parameter schreiben bzw. ändern" vorbereiten und abschicken

     // vom 2. Teilauftrag "Parameter schreiben bzw. ändern" die Antwort abwarten und dann auswerten
     IF #sbRdStart2 THEN

       // Ablöschen des Empfangspuffers
       #sxRespParaMulti.sxHeader.syReqRef := B#16#00;
       #sxRespParaMulti.sxHeader.syReqId := B#16#00;
       #sxRespParaMulti.sxHeader.syAxisNo := B#16#00;
       #sxRespParaMulti.sxHeader.syParaNo := B#16#00;

       FOR #piCount := 1 TO #siLenParaMulti DO
         #sxRespParaMulti.sxData[#piCount] := B#16#00;
       END_FOR;

       // LESEN AZYKLISCH
       #piLenTele := #siLenHeader + #siLenParaMulti;
       #RDREC_1(REQ := True,                                // Startimpuls
                ID := #hardwareId,                         // Diagnoseadresse        
                INDEX := 47,                                  // Rahmentyp           
                MLEN := INT_TO_UINT(#piLenTele),             // maximale Länge
                VALID => #pbValidSFB,                         // neuer Datensatz empfangen und gültig   
                BUSY => #sbRdBusy,                           // Slave beschäftigt
                ERROR => #sbRdError,                          // Fehler beim Schreiben
                STATUS => #pdStatus,                           // Status[1] = Error => Status[2] Error Decode + Status[3] Error Code 
                LEN => #piLenSFB,                           // Länge des gelesenen Datensatzes
                RECORD := #sxRespParaMulti);                   // Zeiger auf gelesenen Datensatz

       // Ausgänge setzen
       #sbBusy := #sbRdBusy;
       #sbDone := #pbValidSFB;

       // Fehler auswerten
       IF #sbRdError THEN
         // Fehlerstatus aus dem Doppelwort filtern und weitergeben                
         #pwWord1 := DWORD_TO_WORD(SHR(IN := (#pdStatus AND DW#16#FFFF00), N := 8));

         // Fehlerstatus setzen
         #siErrorId := 3;
         #DiagId := #pwWord1;

         //Temporärer Fehler: #pdStatus = 80A7, 80B5, 80C0, 80C1, 80C2, 80C3 oder 80C4 zulassen und nocheinmal versuchen
         IF NOT (#pwWord1 = DW#16#80A7) AND NOT (#pwWord1 = DW#16#80B5) AND NOT (#pwWord1 = DW#16#80C0) AND
           NOT (#pwWord1 = DW#16#80C1) AND NOT (#pwWord1 = DW#16#80C2) AND NOT (#pwWord1 = DW#16#80C3) AND
           NOT (#pwWord1 = DW#16#80C4) THEN

           // Wiederholungsauftrag wieder zurücknehmen
           #sbWrStart2 := False;
           #sbRdStart2 := False;
           #sbWrite := False;

           // Fehler ausgeben 
           #sbError := #sbRdError;

         ELSE
           // Fehlerwiederholauftrag ??                   
           IF #siErrorCount = #siMaxErrCount THEN

             // Wiederholungsauftrag wieder zurücknehmen
             #sbWrStart2 := False;
             #sbRdStart2 := False;
             #sbWrite := False;

             //Fehlerzähler zurücksetzen
             #siErrorCount := 0;


             // Fehler ausgeben 
             #sbError := #sbRdError;

             // nix tun bis Zähler überläuft
           ELSE
             #siErrorCount := #siErrorCount + 1;
           END_IF;
         END_IF;

         // Fehler : die Auftragsreferenz der Antwort übertimmt nicht mit der Auftragsreferenz der Anfrage überein
       ELSIF NOT (#siReqRef = BYTE_TO_INT(#sxRespParaMulti.sxHeader.syReqRef)) AND NOT #sbRdBusy AND #pbValidSFB THEN
         #siErrorId := 1;
         #sbError := True;
         #sbDone := False;

         // Wiederholungsauftrag wieder zurücknehmen
         #sbWrStart2 := False;
         #sbRdStart2 := False;
         #sbWrite := False;

         // Fehler : falsche Auftragskennung zurück erhalten    
       ELSIF NOT (#sxRespParaMulti.sxHeader.syReqId = B#16#82 OR #sxRespParaMulti.sxHeader.syReqId = B#16#02) AND
         NOT #sbRdBusy AND #pbValidSFB THEN
         #siErrorId := 1;
         #sbError := True;
         #sbDone := False;

         // Wiederholungsauftrag wieder zurücknehmen
         #sbWrStart2 := False;
         #sbRdStart2 := False;
         #sbWrite := False;

         // Fehler : die angeforderte Anzahl Parameter entspricht nicht der übermittelten Anzahl Parameter überein
       ELSIF NOT (#sxRespParaMulti.sxHeader.syParaNo = B#16#01) AND NOT #sbRdBusy AND #pbValidSFB THEN
         #siErrorId := 1;
         #sbError := True;
         #sbDone := False;

         // Wiederholungsauftrag wieder zurücknehmen
         #sbWrStart2 := False;
         #sbRdStart2 := False;
         #sbWrite := False;

         // Fehler : die Achse entspricht nicht der übergebenen Achse
       ELSIF NOT (#syAxisNo = #sxRespParaMulti.sxHeader.syAxisNo) AND NOT #sbRdBusy AND #pbValidSFB THEN
         #siErrorId := 1;
         #sbError := True;
         #sbDone := False;

         // Wiederholungsauftrag wieder zurücknehmen
         #sbWrStart2 := False;
         #sbRdStart2 := False;
         #sbWrite := False;

         // kein Fehler beim LESEN AZYKLISCH und Auftrag fertig 
       ELSIF NOT #sbRdBusy AND #pbValidSFB THEN

         // 2. Teilauftrag "Parameter schreiben bzw. ändern" negative Rückmeldung erhalten 
         IF #sxRespParaMulti.sxHeader.syReqId = B#16#82 THEN

           // die angefragten Parameter auswerten und im Puffer abspeichern
           // Format des Parameters auswerten, bei Format = Error Fehler auswerten 
           IF (BYTE_TO_INT(#sxRespParaMulti.sxData[1]) = 68) THEN

             // Fehlerwert ermitteln und abspeichern 
             // Format = Word, zwei Bytes zu übermitteltem Parameterwert zusammenfassen
             #pwWordHigh := SHL(IN := BYTE_TO_WORD(#sxRespParaMulti.sxData[3]), N := 8);
             #pwWordLow := BYTE_TO_WORD(#sxRespParaMulti.sxData[4]);
             #pwWord1 := #pwWordHigh XOR #pwWordLow;

             #sbError := True;

             // ermittelte Fehlernummer im Puffer zurücksetzen
             #ErrorNo := W#16#00;

             #ErrorNo := #pwWord1;

             // Die Fehlerhaftigkeit des erkannten Parameter in der Fehlernummer eintragen   
             #swParaError := #swParaError OR W#16#01;

           ELSE

             // Die Fehlerhaftigkeit des erkannten Parameter in der Fehlernummer löschen   
             #swParaError := #swParaError AND W#16#FFFE;

             // ermittelte Fehlernummer im Puffer zurücksetzen
             #ErrorNo := W#16#00;
           END_IF;
         END_IF; // 2. Teilauftrag "Parameter schreiben bzw. ändern" negative Rückmeldung erhalten

         // Fehlerkennung zurücknehmen
         IF (#siErrorId = 3) OR (#siErrorId = 1) THEN
           #siErrorId := 0;
           #sbError := False;
         END_IF;

         #DiagId := W#16#00;

         // 2. Teilauftrag "Parameter schreiben bzw. ändern" ist abgeschlossen
         #sbRdStart2 := False;
         #sbWrite := False;

       END_IF; // kein Fehler beim LESEN AZYKLISCH und Auftrag fertig 
     END_IF; // vom 2. Teilauftrag "Parameter schreiben bzw. ändern" die Antwort abwarten und dann auswerten 
   END_IF; // Auftrag "Parameter schreiben" wurde ausgelöst

   #pdDWordHigh := SHL(IN := INT_TO_DWORD(#siErrorId), N := 16);
   #pdDWordLow := WORD_TO_DWORD(#swParaError);

   // ermittelter Parameterwert eintragen (Word)
   #ErrorId := #pdDWordHigh XOR #pdDWordLow;

   // Initialisierung von Ausgängen
   #Busy := #sbBusy;
   #Error := #sbError;
   #Format := #syFormat;
   // Änderung wegen verhalten von Ready  
   #Done := #sbDone;
   // Prüfen, ob Auftrag abgeschlossen ist
   IF ((#Error OR #Done) AND NOT #sbReady) THEN
     #Ready := True;
     #sbReady := True;
   ELSE
     #Ready := False;
   END_IF;
END_FUNCTION_BLOCK

// ===== library: MasterCopy "SINA_SPEED" =====

FUNCTION_BLOCK "SINA_SPEED"   // FB285, SCL
TITLE = 'Speed Control with SINAMICS and S7'
{ S7_Optimized_Access := 'TRUE' }
AUTHOR : DRVDPS7
FAMILY : DRIVES
NAME : SINA_SPD
VERSION : 5.1
// Copyright (C) Siemens AG 2012. All Rights Reserved. Confidential
// -------------------------------------------------------------------------------------- 
// SINA_SPEED: Drehzahlregelung mit dem Antriebsbaustein SINAMICS S120/G120 <-> S7-1200
// ------------------------------------------------------------------------------------- Ersteller: Siemens AG Erlangen A&D MC PM   Datum:  07.07.10        Vers.:2.1
// Änderung:  J.B. Typical Team                       07.12.12              2.2
//     Umsetzung in SCL / TIA 
// Änderung:  J.B. Typical Team                       29.04.13              2.3
//     1. "Q" an den AusgÃ¤nge entfernen
//     2. Neuer Ausgang PwrInhibit
// Änderung:  J.B. Typical Team                       28.06.13              2.4
//     Ã„nderung HW-Zugriff Ã¼ber LOG2MOD
//      
// Änderung:  J.B. Typical Team                       18.07.13              2.5
//     Ã„nderung HW-Zugriff Ã¼ber zwei HW-EingÃ¤nge
// 
// Änderung:  J.B. Typical Team                       17.07.14              3.0
//     Optimmierung
// 
// Änderung:  J.B. Typical Team                       30.07.14              4.0
//     Festlegung auf einheitlicher neuer Version 4.0
// 
// Änderung:  P.Z. Typical Team                       03.12.15              4.1
//     Schnittstelle an Programmierleitfadeb TIA-Potal angepasst
//     zusÃ¤tzlicher Eingang "ConfigAxis" fÃ¼r STW-Bits
// 
// Änderung:  G.F. Typical Team                       01.03.16              4.2
//     Sollwert auf INT - Grenzen begrenzt
// Änderung:  F.G. Typical Team                       13.09.16              4.3
//     Ausgabewerte am Ausgang "Status" angepasst 
// 
// Änderung:  G.F. Typical Team                       11.01.17              5.0
//     - Festlegung auf einheitlicher neuer Version 5.0 
// 
// Änderung:  G.F. Typical Team                       03.05.18              5.1
//     - Alle Bits des Eingang ConfigAxis auf STW1 aufgelegt 
// 
// Bibliothek V7
// Funktion: Drehzahlregelung mit dem Antriebsbaustein SINAMICS S120/G120 <-> S7-1200
// ********************************************************************************************************************************************************
// ************************************************************************FB283***************************************************************************
// ********************************************************************************************************************************************************
// Copyright (C) Siemens AG 2012. All Rights Reserved. Confidential
// -------------------------------------------------------------------------------------- 
// SINA_SPEED: Drehzahlregelung mit dem Antriebsbaustein SINAMICS S120/G120 <-> S7-1200
// ------------------------------------------------------------------------------------- Ersteller: Siemens AG Erlangen A&D MC PM   Datum:  07.07.10        Vers.:2.1
// Ã„nderung:  J.B. Typical Team                       07.12.12              2.2
//     Umsetzung in SCL / TIA 
// Ã„nderung:  J.B. Typical Team                       29.04.13              2.3
//     1. "Q" an den AusgÃ¤nge entfernen
//     2. Neuer Ausgang PwrInhibit
// Ã„nderung:  J.B. Typical Team                       28.06.13              2.4
//     Ã„nderung HW-Zugriff Ã¼ber LOG2MOD
//      
// Ã„nderung:  J.B. Typical Team                       18.07.13              2.5
//     Ã„nderung HW-Zugriff Ã¼ber zwei HW-EingÃ¤nge
// 
// Ã„nderung:  J.B. Typical Team                       17.07.14              3.0
//     Optimmierung
// 
// Ã„nderung:  J.B. Typical Team                       30.07.14              4.0
//     Festlegung auf einheitlicher neuer Version 4.0
// 
// Ã„nderung:  P.Z. Typical Team                       03.12.15              4.1
//     Schnittstelle an Programmierleitfadeb TIA-Potal angepasst
//     zusÃ¤tzlicher Eingang "ConfigAxis" fÃ¼r STW-Bits
// 
// Ã„nderung:  G.F. Typical Team                       01.03.16              4.2
//     Sollwert auf INT - Grenzen begrenzt
// Ã„nderung:  F.G. Typical Team                       13.09.16              4.3
//     Ausgabewerte am Ausgang "Status" angepasst 
// 
// Ã„nderung:  G.F. Typical Team                       11.01.17              5.0
//     - Festlegung auf einheitlicher neuer Version 5.0 
// 
// Ã„nderung:  G.F. Typical Team                       03.05.18              5.1
//     - Alle Bits des Eingang ConfigAxis auf STW1 aufgelegt 
// 
// Bibliothek V7
// Funktion: Drehzahlregelung mit dem Antriebsbaustein SINAMICS S120/G120 <-> S7-1200
// ********************************************************************************************************************************************************
// ************************************************************************FB283***************************************************************************
// ********************************************************************************************************************************************************
   VAR_INPUT
      EnableAxis : Bool := 0;   // 0-->1; 1 = Enable the drive (OFF2 / OFF 3 are 1 in default status) (OFF1 = 0-->1) / 0-->1 = Einschalten des Antriebs (OFF1 = 0-->1)
      AckError : Bool := 0;   // 1 = Acknowledge drive error / 1 = Fehlerquitierung angestoßen
      SpeedSp : Real := 0.0;   // Speed standardises with the standardisation factor / Drehzahlsollwert [rpm]
      RefSpeed : Real := 0.0;   // Standardisation factor of speed / Referenzdrehzahl (p2000 in [rpm])
      ConfigAxis : Word := 16#003F;   // binary programmed input to control all functions in the telegram without its own function block input / Binärcodierter Eingang zur Ansteuerung aller nicht als Bausteineingang verfügbaren Steuerbits
      HWIDSTW : HW_IO := 0;   // Hardware Identifer set point slot / Hardware Identifer des Sollwert Slots
      HWIDZSW : HW_IO := 0;   // Hardware Identifer actual value slot / Hardware Identifer des Istwert Slots
   END_VAR
   VAR_OUTPUT
      AxisEnabled : Bool := 0;   // 1 = Drive is enabled / 1 = Antrieb in Betrieb
      Lockout : Bool := 0;   // 1 = Drive lockout active / 1 = Einschaltsperre aktiv
      ActVelocity : Real := 0.0;   // Actual in [U/min] / Aktuelle Geschwindigkeit [rpm]
      Error : Bool := 0;   // 1 = Error (FB and Infeed) / 1 = Fehler im Baustein / Antrieb
      Status : Word := 0;   // Status output (7002 = FB in operation; 8xxx = error description - read the manual) / Statusausgabe (7002 = FB in Betrieb; 8xxx = Feherbeschreibung siehe Doku)
      DiagId : Word := 16#0000;   // Error codes of the cyclic system funtion blocks DPWR / DPRD_DAT / Fehlercode der zyklischen Systemfunktionen DPWR / DPRD_DAT
   END_VAR
   VAR
      sxSendBuf : Struct   // Send buffer
         STW1 : Word := WORD#16#0000;   // STW1sxSTW1 : STRUCT Bit08 : BOOL:=False; // ST-Wort-1 Bit 08 --> Reserve Bit09 : BOOL:=False; // ST-Wort-1 Bit 09 --> Reserve Bit10 : BOOL:=True; // ST-Wort-1 Bit 10 --> FÃ¼hrung durch PLC Dir : BOOL:=False; // ST-Wort-1 Bit 11 --> Direction Bit12 : BOOL:=False; // ST-Wort-1 Bit 12 --> Haltebremse unbedingt Ã¶ffnen Bit13 : BOOL:=False; // ST-Wort-1 Bit 13 --> Motorpotenziometer Sollwert hÃ¶her Bit14 : BOOL:=False; // ST-Wort-1 Bit 14 --> Motorpotenziometer Sollwert tiefer Bit15 : BOOL:=False; // ST-Wort-1 Bit 15 --> Reserviert Off1 : BOOL:=False; // ST-Wort-1 Bit 00 --> OFF1/ON (flanks acceptance) Off2 : BOOL:=True; // ST-Wort-1 Bit 01 --> OFF2/ON (enable possible) Off3 : BOOL:=True; // ST-Wort-1 Bit 02 --> OFF3/ON (enable possible) InvEn : BOOL:=True; // ST-Wort-1 Bit 03 --> Enable controller RampEn : BOOL:=True; // ST-Wort-1 Bit 04 --> Ramp enable RampOn : BOOL:=True; // ST-Wort-1 Bit 05 --> Ramp On SpEn : BOOL:=True; // ST-Wort-1 Bit 06 --> Speed set point enable AckFlt : BOOL:=False; // ST-Wort-1 Bit 07 --> Acknowledge fault END_STRUCT;
         Velocity : Word := WORD#16#0000;   // Setpoint of velocity
      END_STRUCT;
      sxRecvBuf : Struct   // Receive buffer
         ZSW1 : Word := WORD#16#0000;   // ZSW1sxZSW1 : STRUCT SpDev : BOOL:=False; // ZSW-Wort-1 = Schleppfehler im Toleranzbereich Pcd : BOOL:=False; // ZSW-Wort-1 = PZD-FÃ¼hrung erreicht Comp : BOOL:=False; // ZSW-Wort-1 = Zielposition erreicht CurLim : BOOL:=False; // ZSW-Wort-1 = Referenzpunkt gesetzt Brake : BOOL:=False; // ZSW-Wort-1 = Haltebremse Ã¶ffnen Motover : BOOL:=False; // ZSW-Wort-1 = keine Warnung Ãœbertemperatur Motor Dir : BOOL:=False; // ZSW-Wort-1 = Direction Invover : BOOL:=False; // ZSW-Wort-1 = keine Warnung thermische Ãœberlast Leistungsteil Rts : BOOL:=False; // ZSW-Wort-1 = Ready to power up / to start Rdy : BOOL:=False; // ZSW-Wort-1 = Ready to operate IOp : BOOL:=False; // ZSW-Wort-1 = In operation (operation enabled) Fault : BOOL:=False; // ZSW-Wort-1 = Fault present NoOff2 : BOOL:=False; // ZSW-Wort-1 = OFF2 inactive NoOff3 : BOOL:=False; // ZSW-Wort-1 = OFF3 inactive Inhibit : BOOL:=False; // ZSW-Wort-1 = Power ON inhibit active Alarm : BOOL:=False; // ZSW-Wort-1 = Alarm / Warning present END_STRUCT;
         Velocity : Word := WORD#16#0000;   // Feedback of velocity
      END_STRUCT;
   END_VAR
   VAR_TEMP
      piRetSFC : Int;   // Status for fault analysis
      piCount : Int;   // Freely available counter variable 3
      prVelocity : Real;   // velocity
      pdRecvBuf : DWord;   // Buffer of Recv-Value
      pdSendBuf : DWord;   // Buffer of Send-Value
      phLAddr : HW_IO;   // Start addr from the I/O process image area of mod (DEC) for DPWR_DAT/DPRD_DAT / Adresse des Sollwert Slots
      swSendBuf : Array[0..1] of Word;   // Sendepuffer
      swRecvBuf : Array[0..1] of Word;   // Empfangspuffer Static variables
   END_VAR
BEGIN

   //=============================================================================
   //SIEMENS AG
   //(c)Copyright 2017 All Rights Reserved
   //-----------------------------------------------------------------------------
   // Library: DriveLib
   // Tested with: S7-1516-3 PN/DP V1.8
   // Engineering: TIA Portal V14
   // Restrictions: -
   // Requirements: S7-1200 / S7-1500
   // Functionality: cyclic communication between a SINAMICS a PLC.
   //                If in HWConfig Std.TLG 1 is projected 2 PZD-words are exchanged
   //                in every bus cycle.
   //                The parametrisation of these words is described in the manual of the
   //                SINAMICS
   //=============================================================================

   // Schreibdaten zusammenstellen
   // Steuerword aufbereiten

   #sxSendBuf.STW1.%X0 := #EnableAxis;
   #sxSendBuf.STW1.%X1 := #ConfigAxis.%X0;
   #sxSendBuf.STW1.%X2 := #ConfigAxis.%X1;
   #sxSendBuf.STW1.%X3 := #ConfigAxis.%X2;
   #sxSendBuf.STW1.%X4 := #ConfigAxis.%X3;
   #sxSendBuf.STW1.%X5 := #ConfigAxis.%X4;
   #sxSendBuf.STW1.%X6 := #ConfigAxis.%X5;
   #sxSendBuf.STW1.%X7 := #AckError;
   #sxSendBuf.STW1.%X8 := #ConfigAxis.%X10;
   #sxSendBuf.STW1.%X9 := #ConfigAxis.%X11;
   #sxSendBuf.STW1.%X10 := TRUE;
   #sxSendBuf.STW1.%X11 := #ConfigAxis.%X6;
   #sxSendBuf.STW1.%X12 := #ConfigAxis.%X7;
   #sxSendBuf.STW1.%X13 := #ConfigAxis.%X8;
   #sxSendBuf.STW1.%X14 := #ConfigAxis.%X9;
   #sxSendBuf.STW1.%X15 := #ConfigAxis.%X12;

   // Geschwindigkeit
   IF #RefSpeed <> 0 THEN
     #prVelocity := #SpeedSp * (16384.0 / #RefSpeed);
     // Limit REAL - Variable to INT - Limits
     IF #prVelocity > 32767 THEN
       #prVelocity := 32767;
     ELSIF #prVelocity < -32768 THEN
       #prVelocity := -32768;
     ELSE
       ; // not needed
     END_IF;
     #sxSendBuf.Velocity := INT_TO_WORD(REAL_TO_INT(#prVelocity));

   ELSE
     #sxSendBuf.Velocity := W#16#0;
   END_IF;
   #swSendBuf[0] := #sxSendBuf.STW1;
   #swSendBuf[1] := #sxSendBuf.Velocity;

   //Prozessdaten zur Signalbaugruppe schreiben
   #piRetSFC := DPWR_DAT(LADDR := #HWIDSTW,
                         RECORD := #swSendBuf);

   // Fehler der RÃ¼ckmeldung ausgeben
   #DiagId := INT_TO_WORD(#piRetSFC);

   //kein Fehler beim Schreiben
   IF #piRetSFC = 0 THEN

     //kein Fehler beim Schreiben
     IF #piRetSFC = 0 THEN

       //Prozessdaten von der Signalbaugruppe lesen
       #piRetSFC := DPRD_DAT(LADDR := #HWIDZSW,
                             RECORD => #swRecvBuf);

       // Fehler der RÃ¼ckmeldung ausgeben
       #DiagId := INT_TO_WORD(#piRetSFC);
     END_IF;

     //Fehler beim Lesen (Profibus-Kommunikation unterbrochen)
     IF #piRetSFC <> 0 THEN

       // Fehler
       #Error := TRUE;
       #Status := 16#8600;

       // Zustandsworte lÃ¶schen
       #sxRecvBuf.ZSW1.%X8 := 0;
       #sxRecvBuf.ZSW1.%X9 := 0;
       #sxRecvBuf.ZSW1.%X10 := 0;
       #sxRecvBuf.ZSW1.%X11 := 0;
       #sxRecvBuf.ZSW1.%X12 := 0;
       #sxRecvBuf.ZSW1.%X13 := 0;
       #sxRecvBuf.ZSW1.%X14 := 0;
       #sxRecvBuf.ZSW1.%X15 := 0;
       #sxRecvBuf.ZSW1.%X0 := 0;
       #sxRecvBuf.ZSW1.%X1 := 0;
       #sxRecvBuf.ZSW1.%X2 := 0;
       #sxRecvBuf.ZSW1.%X3 := 0;
       #sxRecvBuf.ZSW1.%X4 := 0;
       #sxRecvBuf.ZSW1.%X5 := 0;
       #sxRecvBuf.ZSW1.%X6 := 0;
       #sxRecvBuf.ZSW1.%X7 := 0;


       (*#sxRecvBuf.sxZSW1.SpDev   := 0;
       #sxRecvBuf.sxZSW1.Pcd     := 0;
       #sxRecvBuf.sxZSW1.Comp    := 0;
       #sxRecvBuf.sxZSW1.CurLim  := 0;
       #sxRecvBuf.sxZSW1.Brake   := 0;
       #sxRecvBuf.sxZSW1.Motover := 0;
       #sxRecvBuf.sxZSW1.Dir     := 0;
       #sxRecvBuf.sxZSW1.Invover := 0;
       #sxRecvBuf.sxZSW1.Rts     := 0;
       #sxRecvBuf.sxZSW1.Rdy     := 0;
       #sxRecvBuf.sxZSW1.IOp     := 0;
       #sxRecvBuf.sxZSW1.Fault   := 0;
       #sxRecvBuf.sxZSW1.NoOff2  := 0;
       #sxRecvBuf.sxZSW1.NoOff3  := 0;
       #sxRecvBuf.sxZSW1.Inhibit := 0;
       #sxRecvBuf.sxZSW1.Alarm   := 0;*)

       #sxRecvBuf.Velocity := W#16#00;

       // Werte auslesen
     ELSE
       #sxRecvBuf.ZSW1 := #swRecvBuf[0];
       #sxRecvBuf.Velocity := #swRecvBuf[1];

       // ZSW1 aufbereiten                       
       #AxisEnabled := #sxRecvBuf.ZSW1.%X2;
       #Error := #sxRecvBuf.ZSW1.%X3 OR #sxRecvBuf.ZSW1.%X6;
       #Lockout := #sxRecvBuf.ZSW1.%X6;

       // Fehler auswerten
       IF #sxRecvBuf.ZSW1.%X3 THEN
         #Status := 16#8401;
       ELSIF #sxRecvBuf.ZSW1.%X6 THEN
         #Status := 16#8402;
       ELSE
         #Status := 16#7002;
       END_IF;

       (*#Busy       := #sxRecvBuf.sxZSW1.IOp;
       #Error      := #sxRecvBuf.sxZSW1.Fault OR #sxRecvBuf.sxZSW1.Inhibit;
       #PwrInhibit := #sxRecvBuf.sxZSW1.Inhibit;            

       // Fehler auswerten
       IF #sxRecvBuf.sxZSW1.Fault THEN
           #ErrorId := 1;
       ELSIF #sxRecvBuf.sxZSW1.Inhibit THEN 
           #ErrorId := 2;
       ELSE
           #ErrorId := 0;    
       END_IF;*)

       // Geschwindigkeit
       IF #RefSpeed <> 0 THEN
         #ActVelocity := INT_TO_REAL(WORD_TO_INT(#sxRecvBuf.Velocity)) / (16384.0 / #RefSpeed);
       ELSE
         #ActVelocity := 0.0;
       END_IF;
     END_IF;
   ELSE

     // Fehler
     #Error := TRUE;
     #Status := 16#8601;

   END_IF;
END_FUNCTION_BLOCK

// ===== library: MasterCopy "SINA_POS" =====

FUNCTION_BLOCK "SINA_POS"   // FB284, SCL
TITLE = 'Positioning with SINAMICS and S7'
{ S7_Optimized_Access := 'TRUE' }
AUTHOR : DRVDPS7
FAMILY : DRIVES
NAME : SINA_POS
VERSION : 5.7
// Copyright (C) Siemens AG 2012. All Rights Reserved. Confidential
// -------------------------------------------------------------------------------------- 
// SINA_POS: Positionierung mit dem Antriebsbaustein SINAMICS S120/G120 <-> S7-1200
// ------------------------------------------------------------------------------------- Ersteller: Siemens AG Erlangen A&D MC PM   Datum:  07.07.10        Vers.:2.1
// Änderung:  J.B. Typical Team                       18.12.12              2.2
//     Umsetzung in SCL / TIA 
// Änderung:  J.B. Typical Team                       18.04.13              2.3
//     Bei Betriebsart "Referenzieren - Referenzpunkt setzen"
//     nicht intern setzen sondern Eingang #Execute abfragen als 
//     Startbedingung
// Änderung:  J.B. Typical Team                       29.04.13              2.4
//     1. Off1 möglich bei ungültige Betriebsart
//     2. Referenzpunkt setzen Exceute übernehmen
//     3. Fehlermeldung ausgeben bei Wechel ohne 
//        Beendigung der Betriebsart 
//     4. "Q" an den Ausgänge entfernen
//     5. Neuer Ausgang PwrInhibit
//      
// Änderung:  J.B. Typical Team                       14.05.13              2.5
//     Fehlerbehebung und Defaultwerte ändern
// Änderung:  J.B. Typical Team                       28.06.13              2.6
//     HW-Zugriffsermittlung über LOG2MOD
// Änderung:  J.B. Typical Team                       18.07.13              2.7
//     HW-Zugriffsermittlung über zwei HW-Eingänge
// Änderung:  J.B. Typical Team                       18.09.13              2.8
//     Konvertierungsfehler behoben
// Änderung:  J.B. Typical Team                       25.09.13              2.9
//     Bei Betriebswechsel von 3 nach 6 darf MidStart nicht sitzen
// Änderung:  J.B. Typical Team                       31.03.14              3.0
//     In der Betriebsart 1-3 und 6 darf MidTrTyp nicht sitzen
// Änderung:  J.B. Typical Team                       25.06.14              3.1
//     Das Quittierbit "AckFlt" immer durchreichen
// Änderung:  J.B. Typical Team                       30.07.14              4.0
//     Festlegung auf einheitlicher neuer Version 4.0
// Änderung:  J.B. Typical Team                       07.11.14              4.1
//     Fehlerbehebung falsche Zuweisung von Off1 bei Mode 4
//     und Mode 8(DriveLib V4 - RQ 346046)
// Änderung:  F.G. Typical Team                       16.04.15              4.2
//     Anzahl der Zyklen die auf die Rückmeldung fliegendes Ref.
//     gewartet wird verdoppelt (siRetryMax = 10)  (DriveLib V4 - RQ 367986)
// Änderung:  F.G. Typical Team                       15.09.15              4.3
//     Anzahl der Zyklen die auf die Rückmeldung fliegendes Ref.
//     gewartet noch einmal um 5 erhöht (siRetryMax = 15)  (DriveLib V4 - RQ 367986)
// Änderung:  F.G. Typical Team                       15.09.15              4.4
//     Abfrage des richtigen Bits im EPosZSW1 (Zeile 1394)es muss das Bit12 
//     und nicht das Bit 11 abgefragt werden  (DriveLib V4 - RQ 367986)
// Änderung:  F.G. Typical Team                       03.12.15              4.5
//     1. Ein-/Ausgänge an Programmierleitfaden für TIA-Portal angepasst
//        Zusätzlicher Eingang um alle Bits in den STWs zu bedienen
//     2. Warnung durch Initialisierung elimininiert
// Änderung:  F.G. Typical Team                       13.09.16              4.6
//     Ausgabewerte am Ausgang "Status" angepasst 
// 
// Änderung:  G.F. Typical Team                       11.01.17              5.0
//     - Festlegung auf einheitlicher neuer Version 5.0 
// 
// Änderung:  G.F. Typical Team                       13.07.17              5.1
//     - Zuordnung der Bits von ConfigPos korrigiert 
// 
// Änderung:  G.F. Typical Team                       12.01.18              5.2
//     - RQ2637983 sxSendBuf.EPosSTW2.%X1 in Mode 7 und 8 rücksetzen 
// Änderung:  G.F. Typical Team                       20.07.18              5.3
//     - ZSW1.13 als Ausgang zur Verfügung gestellt (wegen FW - Änderung)
// Änderung:  G.F. Typical Team                       18.10.18              5.4
//     - RQ 824321 Zähler für fliegendes Referenzieren zurücksetzen
// Änderung:  G.F. Typical Team                       08.02.19              5.5
//     - Version wegen Änderungen in älteren Lib-Versionen 
// Änderung:  G.F. Typical Team                       08.02.19              5.6
//     - RQ 3901129 Fehler Flankenauswertung Eingang ExecuteMode behoben Bibliothek V7
// Änderung:  G.F. Typical Team                       17.05.19              5.7
//     - RQ 4094299 Fehler Referenzfahrt wird nicht gestartet behoben Bibliothek V7
// Funktion: Positionierung mit dem Antriebsbaustein SINAMICS S120/G120 <-> S7-1200
// ********************************************************************************************************************************************************
// ************************************************************************FB283***************************************************************************
// ********************************************************************************************************************************************************
// Copyright (C) Siemens AG 2012. All Rights Reserved. Confidential
// -------------------------------------------------------------------------------------- 
// SINA_POS: Positionierung mit dem Antriebsbaustein SINAMICS S120/G120 <-> S7-1200
// ------------------------------------------------------------------------------------- Ersteller: Siemens AG Erlangen A&D MC PM   Datum:  07.07.10        Vers.:2.1
// Änderung:  J.B. Typical Team                       18.12.12              2.2
//     Umsetzung in SCL / TIA 
// Änderung:  J.B. Typical Team                       18.04.13              2.3
//     Bei Betriebsart "Referenzieren - Referenzpunkt setzen"
//     nicht intern setzen sondern Eingang #Execute abfragen als 
//     Startbedingung
// Änderung:  J.B. Typical Team                       29.04.13              2.4
//     1. Off1 möglich bei ungültige Betriebsart
//     2. Referenzpunkt setzen Exceute übernehmen
//     3. Fehlermeldung ausgeben bei Wechel ohne 
//        Beendigung der Betriebsart 
//     4. "Q" an den Ausgänge entfernen
//     5. Neuer Ausgang PwrInhibit
//      
// Änderung:  J.B. Typical Team                       14.05.13              2.5
//     Fehlerbehebung und Defaultwerte ändern
// Änderung:  J.B. Typical Team                       28.06.13              2.6
//     HW-Zugriffsermittlung über LOG2MOD
// Änderung:  J.B. Typical Team                       18.07.13              2.7
//     HW-Zugriffsermittlung über zwei HW-Eingänge
// Änderung:  J.B. Typical Team                       18.09.13              2.8
//     Konvertierungsfehler behoben
// Änderung:  J.B. Typical Team                       25.09.13              2.9
//     Bei Betriebswechsel von 3 nach 6 darf MidStart nicht sitzen
// Änderung:  J.B. Typical Team                       31.03.14              3.0
//     In der Betriebsart 1-3 und 6 darf MidTrTyp nicht sitzen
// Änderung:  J.B. Typical Team                       25.06.14              3.1
//     Das Quittierbit "AckFlt" immer durchreichen
// Änderung:  J.B. Typical Team                       30.07.14              4.0
//     Festlegung auf einheitlicher neuer Version 4.0
// Änderung:  J.B. Typical Team                       07.11.14              4.1
//     Fehlerbehebung falsche Zuweisung von Off1 bei Mode 4
//     und Mode 8(DriveLib V4 - RQ 346046)
// Änderung:  F.G. Typical Team                       16.04.15              4.2
//     Anzahl der Zyklen die auf die Rückmeldung fliegendes Ref.
//     gewartet wird verdoppelt (siRetryMax = 10)  (DriveLib V4 - RQ 367986)
// Änderung:  F.G. Typical Team                       15.09.15              4.3
//     Anzahl der Zyklen die auf die Rückmeldung fliegendes Ref.
//     gewartet noch einmal um 5 erhöht (siRetryMax = 15)  (DriveLib V4 - RQ 367986)
// Änderung:  F.G. Typical Team                       15.09.15              4.4
//     Abfrage des richtigen Bits im EPosZSW1 (Zeile 1394)es muss das Bit12 
//     und nicht das Bit 11 abgefragt werden  (DriveLib V4 - RQ 367986)
// Änderung:  F.G. Typical Team                       03.12.15              4.5
//     1. Ein-/Ausgänge an Programmierleitfaden für TIA-Portal angepasst
//        Zusätzlicher Eingang um alle Bits in den STWs zu bedienen
//     2. Warnung durch Initialisierung elimininiert
// Änderung:  F.G. Typical Team                       13.09.16              4.6
//     Ausgabewerte am Ausgang "Status" angepasst 
// 
// Änderung:  G.F. Typical Team                       11.01.17              5.0
//     - Festlegung auf einheitlicher neuer Version 5.0 
// 
// Änderung:  G.F. Typical Team                       13.07.17              5.1
//     - Zuordnung der Bits von ConfigPos korrigiert 
// 
// Änderung:  G.F. Typical Team                       12.01.18              5.2
//     - RQ2637983 sxSendBuf.EPosSTW2.%X1 in Mode 7 und 8 rücksetzen 
// Änderung:  G.F. Typical Team                       20.07.18              5.3
//     - ZSW1.13 als Ausgang zur Verfügung gestellt (wegen FW - Änderung)
// Änderung:  G.F. Typical Team                       18.10.18              5.4
//     - RQ 824321 Zähler für fliegendes Referenzieren zurücksetzen
// Änderung:  G.F. Typical Team                       08.02.19              5.5
//     - Version wegen Änderungen in älteren Lib-Versionen 
// Änderung:  G.F. Typical Team                       08.02.19              5.6
//     - RQ 3901129 Fehler Flankenauswertung Eingang ExecuteMode behoben Bibliothek V7
// Funktion: Positionierung mit dem Antriebsbaustein SINAMICS S120/G120 <-> S7-1200
// ********************************************************************************************************************************************************
// ************************************************************************FB283***************************************************************************
// ********************************************************************************************************************************************************
   VAR_INPUT
      ModePos : Int := 0;   // Settings of the mode / Auswahl EPos Betriebsart (0= keine; 1,2,3 = MDI; 4,5 = Referenzieren; 6= Verfarhsätze; 7,8 = Tippen)
      EnableAxis : Bool := 0;   // 1 = Enable the drive / 0-->1 = Einschalten des Antriebs (OFF1 = 0-->1)
      CancelTraversing : Bool := 1;   // 0 = Reject active traverse task / 0 = Abruch der laufenden Verfahrbewegung (1=kein Abbruch)
      IntermediateStop : Bool := 1;   // 0 = Intermediate STOP of traverse command / 0 = Zwischenhalt der laufenden Verfahrbewegung (1= kein Zwischenhalt)
      Positive : Bool := 0;   // 1 = Direction positive / 1 = Positive Verfahrrichtung
      Negative : Bool := 0;   // 1 = Direction negative / 1 = Negative Verfahrrichtung
      Jog1 : Bool := 0;   // 1 = Use jog 1 (direction / speed) / 1 = Tippen Sollwert 1 auswählen
      Jog2 : Bool := 0;   // 1 = Use jog 2 (direction / speed) / 1 = Tippen Sollwert 2 auswählen
      FlyRef : Bool := 0;   // 1 = Start flying reference function / 1 = Aktivierung Fliegendes Referenzieren (nicht möglich bei ModePos = 4, 5)
      AckError : Bool := 0;   // 1 = Acknowledge of errors / 1 = Achs / EPos Fehlerquittierung anwählen
      ExecuteMode : Bool := 0;   // 0-->1 = Start the mode / 0-->1 = Starten der mit ModePos gewählten Betriebsart
      Position : DInt := 0;   // Position of the MDI mode or setting of traversing block / Positionssollwert [LU] für Direkt Sollwert vorgabe (MDI)
      Velocity : DInt := 0;   // MDI velocity / MDI Geschwindigkeit [1000*LU / min]
      OverV : Int := 100;   // Override of velocity in [%] --> 4000h=100% / Geschwindigkeit Skalierung (Alle Betriebsarten 4000h = 100%))
      OverAcc : Int := 100;   // Override of acceleration in [%] --> 4000h=100% / MDI Beschleunigung (4000h = 100%)
      OverDec : Int := 100;   // Override of deceleration in [%] --> 4000h=100% / MDI Verzögerung (4000h = 100%)
      ConfigEPos : DWord := 16#0000_0003;   // binary programmed input to control all functions in the telegram without its own function block input / Binärcodierter Eingang zur Ansteuerung aller nicht als Bausteineingang verfügbaren Steuerbits
      HWIDSTW : Hw_Io := 0;   // Hardware Identifer set point slot / Hardware Identifer des Sollwert Slots
      HWIDZSW : Hw_Io := 0;   // Hardware Identifer actual value slot / Hardware Identifer des Istwert Slots
   END_VAR
   VAR_OUTPUT
      AxisEnabled : Bool := 0;   // 1= Axis in operation / 1= EPos Achse ist in Betrieb
      AxisPosOk : Bool := 0;   // 1= Position setpoint reached / 1= EPos Achsposition erreicht
      AxisSpFixed : Bool := 0;   // 1= Setpoint fixed (Attention: Dependence on SINAMICS firmware) / 1= Sollwert steht (Achtung: Abhängigkeit von SINAMICS Firmware)
      AxisRef : Bool := 0;   // 1= Reference point set / 1= EPos Achse referenziert
      AxisWarn : Bool := 0;   // 1= Axis alarm / warning present / 1= Antriebswarnung aktiv
      AxisError : Bool := 0;   // 1= Axis fault present / 1= Antriebs / EPos Fehler vorhanden
      Lockout : Bool := 0;   // 1= Axis in lockout state / 1= Einschaltsperre aktiv
      ActVelocity : DInt := 0;   // Actual drive speed (has to be normed with p2000 --> 40000000h = 100%) / Aktuelle Geschwindigkeit (40000000h = 100% von p2000 in [rpm])
      ActPosition : DInt := 0;   // Actual position in [LU] / Aktuelle Position in LU
      ActMode : Int := 0;   // Active EPos mode / Aktuellle Betriebsart
      EPosZSW1 : Word := 0;   // Status of EPOS ZSW1
      EPosZSW2 : Word := 0;   // Status of EPOS ZSW2
      ActWarn : Word := 0;   // Actual number of warning / Aktuelle Warnung
      ActFault : Word := 0;   // Actual number of error / Aktuelle Störung
      Error : Bool := 0;   // 1 = Error (FB and Infeed) / Fehler (Antrieb und / oder Funktionsbaustein)
      Status : Word := 0;   // Status output (7002 = FB in operation; 8xxx = error description - read the manual) / Statusausgabe (7002 = FB in Betrieb; 8xxx = Feherbeschreibung siehe Doku)
      DiagID : Word := 0;   // Error codes of the cyclic system funtion blocks DPWR / DPRD_DAT / Fehlercode der zyklischen Systemfunktionen DPWR / DPRD_DAT
   END_VAR
   VAR
      sbOff1Edge : Bool := 0;   // Positive edge of starting or stopping the device
      sbOff1 : Bool := 0;   // Starting or stopping the device
      sbExecuteEdge : Bool := 0;   // Positive edge of activate traversing block
      sbExecute : Bool := 0;   // Activate traversing block
      sbRefTypEdge : Bool := 0;   // Positive edge of referencing type "flying reference"
      sbRefTyp : Bool := 0;   // Referencing type "flying reference"
      sbMdiStart : Bool := 0;   // Direct setpoint input / MDI - start
      sbMdiStartEdge : Bool := 0;   // Positive edge of direct setpoint input / MDI - start
      sbRefStart : Bool := 0;   // Referencing start
      sbJogInc : Bool := 0;   // Jogging incremental
      sbReady : Bool := 0;   // Ready to power up / to start
      sbIOp : Bool := 0;   // Ready to operate
      sbAccel : Bool := 0;   // Axis accelerating
      sbDecel : Bool := 0;   // Axis decelerating
      sbAlarm : Bool := 0;   // Alarm / Warnung present
      sbFault : Bool := 0;   // Fault present
      sbFWD : Bool := 0;   // Axis drives forwards
      sbBWD : Bool := 0;   // Axis drives backwards
      sbBusy : Bool := 0;   // Mode of operation is explained
      swStatus : Word := 16#0000;   // Mode of operation disturbance
      swEPosZSW1 : Word := 16#0000;   // Status of EPOS ZSW1 / EPos Zustandswort 1
      swEPosZSW2 : Word := 16#0000;   // Status of EPOS ZSW2 / EPos Zustandswort 2
      siExecuteCyc : Int := 0;   // Counter of runcycle of active traversing block
      siRefTypCyc : Int := 0;   // Counter of runcycle of referencing type "flying reference"
      siJogIncCyc : Int := 0;   // Counter of runcycle of jogging incremental
      siMdiStartCyc : Int := 0;   // Counter of runcycle of direct setpoint input / MDI - start
      siRefActRetry : Int := 0;   // Counter of retry of reference point approach active
      siModePos : Int := 0;   // Setting of mode
      siModePosMax : Int := 8;   // Max. count of mode
      siCycWait : Int := 5;   // Counter of cycle of waiting
      siRetryMax : Int := 30;   // Max. count of cycles of retry
      sbModePos : Bool := 0;   // Mode of setting okay
      sxSendBuf : Struct   // send buffer of telegram for sending data to the drive
         STW1 : Word := WORD#16#0000;   // STW1sxSTW1 : STRUCT Jog1 : BOOL:=0; // ST-Wort-1 Bit 08 --> 1 = Jogging - signal source 1 Jog2 : BOOL:=0; // ST-Wort-1 Bit 09 --> 1 = Jogging - signal source 2 LB : BOOL:=1; // Allways // ST-Wort-1 Bit 10 --> 1 = Life bit RefStart : BOOL:=0; // ST-Wort-1 Bit 11 --> 1 = Referencing start / stop Bit12 : BOOL:=0; // ST-Wort-1 Bit 12 --> 1 = Reserve Bit13 : BOOL:=0; // ST-Wort-1 Bit 13 --> 1 = Externer Satzwechsel Bit14 : BOOL:=0; // ST-Wort-1 Bit 14 --> 1 = Reserve Bit15 : BOOL:=0; // ST-Wort-1 Bit 15 --> 1 = Reserve Off1 : BOOL:=0; // ST-Wort-1 Bit 00 --> 1 = OFF1/ON (flanks acceptance) Off2 : BOOL:=1; // Allways // ST-Wort-1 Bit 01 --> 1 = OFF2/ON (enable possible) Off3 : BOOL:=1; // Allways // ST-Wort-1 Bit 02 --> 1 = OFF3/ON (enable possible) Enc : BOOL:=1; // Allways // ST-Wort-1 Bit 03 --> 1 = Enable controller RejTrvTsk : BOOL:=0; // ST-Wort-1 Bit 04 --> 1 = Traversing block and MDI - reject task IntMStop : BOOL:=0; // ST-Wort-1 Bit 05 --> 1 = Traversing block and MDI - intermediate - STOP TrvStart : BOOL:=0; // ST-Wort-1 Bit 06 --> 1 = Traversing start - direct setpoint input / MDI - transfer edge AckFault : BOOL:=0; // ST-Wort-1 Bit 07 --> 1 = Acknowledge fault END_STRUCT;
         EPosSTW1 : Word := WORD#16#0000;   // EPOSSTW1sxEPosSTW1 : STRUCT MdiTyp : BOOL:=0; // EPOS-Wort-1 Bit 08 --> 1 = Direct setpoint input / MDI - positioning type MdiPos : BOOL:=0; // EPOS-Wort-1 BIT 09 --> 1 = Direct setpoint input / MDI - positive direction MdiNeg : BOOL:=0; // EPOS-Wort-1 BIT 10 --> 1 = Direct setpoint input / MDI - negative direction Bit11 : BOOL:=0; // EPOS-Wort-1 BIT 11 --> 1 = Reserve MdiTrTyp : BOOL:=0; // EPOS-Wort-1 BIT 12 --> 1 = Direct setpoint input / MDI - transfer type Bit13 : BOOL:=0; // EPOS-Wort-1 BIT 13 --> 1 = Reserve MdiSetup : BOOL:=0; // EPOS-Wort-1 BIT 14 --> 1 = Direct setpoint input / MDI - setup selection MdiStart : BOOL:=0; // EPOS-Wort-1 BIT 15 --> 1 = Direct setpoint input / MDI - start TrvBit0 : BOOL:=0; // EPOS-Wort-1 BIT 00 --> 1 = Traversing block - block selection bit 0 TrvBit1 : BOOL:=0; // EPOS-Wort-1 BIT 01 --> 1 = Traversing block - block selection bit 1 TrvBit2 : BOOL:=0; // EPOS-Wort-1 BIT 02 --> 1 = Traversing block - block selection bit 2 TrvBit3 : BOOL:=0; // EPOS-Wort-1 BIT 03 --> 1 = Traversing block - block selection bit 3 TrvBit4 : BOOL:=0; // EPOS-Wort-1 BIT 04 --> 1 = Traversing block - block selection bit 4 TrvBit5 : BOOL:=0; // EPOS-Wort-1 Bit 05 --> 1 = Traversing block - block selection bit 5 Bit06 : BOOL:=0; // EPOS-Wort-1 Bit 06 --> 1 = Reserve Bit07 : BOOL:=0; // EPOS-Wort-1 Bit 07 --> 1 = Reserve END_STRUCT;
         EPosSTW2 : Word := WORD#16#0000;   // EPOSSTW2sxEPosSTW2 : STRUCT RefTyp : BOOL:=0; // EPOS-Wort-2 Bit 08 --> 1 = Referencing type RefStDi : BOOL:=0; // EPOS-Wort-2 Bit 09 --> 1 = Homing start direction RefInpS : BOOL:=0; // EPOS-Wort-2 Bit 10 --> 1 = Referencing passive - input selection RefEdge : BOOL:=0; // EPOS-Wort-2 Bit 11 --> 1 = Referencing passive - edge evaluation Bit12 : BOOL:=0; // EPOS-Wort-2 Bit 12 --> 1 = Reserve Bit13 : BOOL:=0; // EPOS-Wort-2 Bit 13 --> 1 = Reserve SftLimAct : BOOL:=0; // EPOS-Wort-2 Bit 14 --> 1 = Software limit switch activation StpCamAct : BOOL:=0; // EPOS-Wort-2 Bit 15 --> 1 = Stop output cam activation TrkMode : BOOL:=0; // EPOS-Wort-2 Bit 00 --> 1 = Tracking mode active SetRefPt : BOOL:=0; // EPOS-Wort-2 Bit 01 --> 1 = Set reference point ActRefCam : BOOL:=0; // EPOS-Wort-2 Bit 02 --> 1 = Reference cam active Bit03 : BOOL:=0; // EPOS-Wort-2 Bit 03 --> 1 = Reserve Bit04 : BOOL:=0; // EPOS-Wort-2 Bit 04 --> 1 = Reserve JogInc : BOOL:=0; // EPOS-Wort-2 Bit 05 --> 1 = Jogging - jogging incremental Bit06 : BOOL:=0; // EPOS-Wort-2 Bit 06 --> 1 = Reserve Bit07 : BOOL:=0; // EPOS-Wort-2 Bit 07 --> 1 = Reserve END_STRUCT;
         STW2 : Word := WORD#16#0000;   // STW2sxSTW2 : STRUCT TrvFixStp : BOOL:=0; // ST-Wort-2 Bit 08 --> 1 = Travel fixed STOP GlbTrgCom : BOOL:=0; // ST-Wort-2 Bit 09 --> 1 = Global trigger command Bit10 : BOOL:=0; // ST-Wort-2 Bit 10 --> 1 = Reserve MotSwOver : BOOL:=0; // ST-Wort-2 Bit 11 --> 1 = Motor switch over finished MsZykBit0 : BOOL:=0; // ST-Wort-2 Bit 12 --> 1 = Master life bit 0 MsZykBit1 : BOOL:=0; // ST-Wort-2 Bit 13 --> 1 = Master life bit 1 MsZykBit2 : BOOL:=0; // ST-Wort-2 Bit 14 --> 1 = Master life bit 2 MsZykBit3 : BOOL:=0; // ST-Wort-2 Bit 15 --> 1 = Master life bit 3 DDSBit0 : BOOL:=0; // ST-Wort-2 Bit 00 --> 1 = Drive data set bit 0 DDSBit1 : BOOL:=0; // ST-Wort-2 Bit 01 --> 1 = Drive data set bit 1 DDSBit2 : BOOL:=0; // ST-Wort-2 Bit 02 --> 1 = Drive data set bit 2 DDSBit3 : BOOL:=0; // ST-Wort-2 Bit 03 --> 1 = Drive data set bit 3 DDSBit4 : BOOL:=0; // ST-Wort-2 Bit 04 --> 1 = Drive data set bit 4 GlbStart : BOOL:=0; // ST-Wort-2 Bit 05 --> 1 = Global start ResIComp : BOOL:=0; // ST-Wort-2 Bit 06 --> 1 = Reset I-component of speed controller ActPrkAxis : BOOL:=0; // ST-Wort-2 Bit 07 --> 1 = Activate parking axis END_STRUCT;
         OverrideV : Word := WORD#16#0000;   // Velocity override
         Position : DWord := DWORD#16#0000_0000;   // Setpoint of position
         Velocity : DWord := DWORD#16#0000_0000;   // Setpoint of velocity
         OverrideA : Word := WORD#16#0000;   // Accelerating override
         OverrideD : Word := WORD#16#0000;   // Decelerating override
         Reserve : Word := WORD#16#0000;   // Reserve
      END_STRUCT;
      sxRecvBuf : Struct   // receive buffer of telegram for receiving data from the drive
         ZSW1 : Word := WORD#16#0000;   // ZSW1sxZSW1 : STRUCT NoFlwErr : BOOL:=0; // ZSW-Wort-1 Bit 08 --> 1 = Following error in tolerance LbCr : BOOL:=0; // ZSW-Wort-1 Bit 09 --> 1 = Lifebit control request TargPos : BOOL:=0; // ZSW-Wort-1 Bit 10 --> 1 = Target position reached RefPSet : BOOL:=0; // ZSW-Wort-1 Bit 11 --> 1 = Reference point set TrvTskAck : BOOL:=0; // ZSW-Wort-1 Bit 12 --> 1 = Traversing task acknowledge StndStill : BOOL:=0; // ZSW-Wort-1 Bit 13 --> 1 = [n_ist] < Drehzahlsollwert 3 Accel : BOOL:=0; // ZSW-Wort-1 Bit 14 --> 1 = Axis accelerating Decel : BOOL:=0; // ZSW-Wort-1 Bit 15 --> 1 = Axis decelerating RTS : BOOL:=0; // ZSW-Wort-1 Bit 00 --> 1 = Ready to power up / to start RDY : BOOL:=0; // ZSW-Wort-1 Bit 01 --> 1 = Ready to operate IOp : BOOL:=0; // ZSW-Wort-1 Bit 02 --> 1 = In operation (operation enabled) Fault : BOOL:=0; // ZSW-Wort-1 Bit 03 --> 1 = Fault present NoOff2Act : BOOL:=0; // ZSW-Wort-1 Bit 04 --> 1 = OFF2 inactive NoOff3Act : BOOL:=0; // ZSW-Wort-1 Bit 05 --> 1 = OFF3 inactive PowInhbt : BOOL:=0; // ZSW-Wort-1 Bit 06 --> 1 = Power ON inhibit active Alarm : BOOL:=0; // ZSW-Wort-1 Bit 07 --> 1 = Alarm / Warning present END_STRUCT;
         EPosZSW1 : Word := WORD#16#0000;   // EPOSZSW1sxEPosZSW1 : STRUCT StpCamMinAct : BOOL:=0; // EPOS-Wort-1 Bit 08 --> 1 = STOP cam minus active StpCamPlsAct : BOOL:=0; // EPOS-Wort-1 Bit 09 --> 1 = STOP cam plus active JogAct : BOOL:=0; // EPOS-Wort-1 Bit 10 --> 1 = Jogging active RefAct : BOOL:=0; // EPOS-Wort-1 Bit 11 --> 1 = Reference point approach active FlyRefAct : BOOL:=0; // EPOS-Wort-1 Bit 12 --> 1 = Flying referencing active TrvBlAct : BOOL:=0; // EPOS-Wort-1 Bit 13 --> 1 = Traversing block active MdiStupAct : BOOL:=0; // EPOS-Wort-1 Bit 14 --> 1 = MDI setup active MdiPosAct : BOOL:=0; // EPOS-Wort-1 Bit 15 --> 1 = MDI positing active ActTrvBit0 : BOOL:=0; // EPOS-Wort-1 BIT 00 --> 1 = Active traversing block bit 0 ActTrvBit1 : BOOL:=0; // EPOS-Wort-1 Bit 01 --> 1 = Active traversing block bit 1 ActTrvBit2 : BOOL:=0; // EPOS-Wort-1 Bit 02 --> 1 = Active traversing block bit 2 ActTrvBit3 : BOOL:=0; // EPOS-Wort-1 Bit 03 --> 1 = Active traversing block bit 3 ActTrvBit4 : BOOL:=0; // EPOS-Wort-1 Bit 04 --> 1 = Active traversing block bit 4 ActTrvBit5 : BOOL:=0; // EPOS-Wort-1 Bit 05 --> 1 = Active traversing block bit 5 Bit06 : BOOL:=0; // EPOS-Wort-1 Bit 06 --> 1 = Reserve Bit07 : BOOL:=0; // EPOS-Wort-1 Bit 07 --> 1 = Reserve END_STRUCT;
         EPosZSW2 : Word := WORD#16#0000;   // EPOSZSW2sxEPosZSW2 : STRUCT PosSmCam1 : BOOL:=0; // EPOS-Wort-2 Bit 08 --> 1 = Position actual value <= cam position 1 PosSmCam2 : BOOL:=0; // EPOS-Wort-2 Bit 09 --> 1 = Position actual value <= cam position 2 TrvOut1 : BOOL:=0; // EPOS-Wort-2 Bit 10 --> 1 = Direct output 1 via traversing block TrvOut2 : BOOL:=0; // EPOS-Wort-2 Bit 11 --> 1 = Direct output 2 via traversing block FxStpRd : BOOL:=0; // EPOS-Wort-2 Bit 12 --> 1 = Fixed STOP reached FxStpTrRd : BOOL:=0; // EPOS-Wort-2 Bit 13 --> 1 = Fixed STOP clamping torque reached TrvFxStpAct : BOOL:=0; // EPOS-Wort-2 Bit 14 --> 1 = Traversing fixed STOP active CmdAct : BOOL:=0; // EPOS-Wort-2 Bit 15 --> 1 = Traversing command active TrkModeAct : BOOL:=0; // EPOS-Wort-2 Bit 00 --> 1 = Tracking mode active VeloLimAct : BOOL:=0; // EPOS-Wort-2 Bit 01 --> 1 = Velocity limit active SetPStat : BOOL:=0; // EPOS-Wort-2 Bit 02 --> 1 = Setpoint static PrnMrkOut : BOOL:=0; // EPOS-Wort-2 Bit 03 --> 1 = Printmark outside outer window FWD : BOOL:=0; // EPOS-Wort-2 Bit 04 --> 1 = Axis forwards BWD : BOOL:=0; // EPOS-Wort-2 Bit 05 --> 1 = Axis backwards SftSwMinAct : BOOL:=0; // EPOS-Wort-2 Bit 06 --> 1 = Software limit switch minus active SftSwPlsAct : BOOL:=0; // EPOS-Wort-2 Bit 07 --> 1 = Software limit switch plus active END_STRUCT;
         ZSW2 : Word := WORD#16#0000;   // ZSW2sxZSW2 : STRUCT Bit08 : BOOL:=0; // ZSW-Wort-2 Bit 08 --> Reserve GlbTrgReq : BOOL:=0; // ZSW-Wort-2 Bit 09 --> Global trigger request PulsEn : BOOL:=0; // ZSW-Wort-2 Bit 10 --> Pulses enabled MotSwOverAct : BOOL:=0; // ZSW-Wort-2 Bit 11 --> Motor switch over activ SlvZykBit0 : BOOL:=0; // ZSW-Wort-2 Bit 12 --> Slave - life bit 0 SlvZykBit1 : BOOL:=0; // ZSW-Wort-2 Bit 13 --> Slave - life bit 1 SlvZykBit2 : BOOL:=0; // ZSW-Wort-2 Bit 14 --> Slave - life bit 2 SlvZykBit3 : BOOL:=0; // ZSW-Wort-2 Bit 15 --> Slave - life bit 3 ActDDSBit0 : BOOL:=0; // ZSW-Wort-2 Bit 00 --> Active drive data set bit 0 ActDDSBit1 : BOOL:=0; // ZSW-Wort-2 Bit 01 --> Active drive data set bit 1 ActDDSBit2 : BOOL:=0; // ZSW-Wort-2 Bit 02 --> Active drive data set bit 2 ActDDSBit3 : BOOL:=0; // ZSW-Wort-2 Bit 03 --> Active drive data set bit 3 ActDDSBit4 : BOOL:=0; // ZSW-Wort-2 Bit 04 --> Active drive data set bit 4 CmdActRelBrk : BOOL:=0; // ZSW-Wort-2 Bit 05 --> Command "release holding break" active TrqContMode : BOOL:=0; // ZSW-Wort-2 Bit 06 --> Torque controlled mode ParkAxisAct : BOOL:=0; // ZSW-Wort-2 Bit 07 --> Parking axis activated END_STRUCT;
         NotUsed : Word := WORD#16#0000;   // Reserve
         Position : DWord := DWORD#16#0000_0000;   // Feedback of position
         Velocity : DWord := DWORD#16#0000_0000;   // Feedback of velocity
         ErrNr : Word := WORD#16#0000;   // Fault number
         WarnNr : Word := WORD#16#0000;   // Warning number
         Reserve : Word := WORD#16#0000;   // Reserve
      END_STRUCT;
   END_VAR
   VAR_TEMP
      piRetSFC : Int;   // Status for fault analysis
      piCount : Int;   // Freely available counter variable 3
      swSendBuf : Array[0..11] of Word;   // Send buffer
      swRecvBuf : Array[0..11] of Word;   // Receive buffer
   END_VAR
BEGIN

